	MoveL Offs(p0,555.9584000000001,76.2912, 0), v100, z5, tool0;
	MoveL Offs(p0,560.0348,77.80539999999999, 0), v100, z5, tool0;
	MoveL Offs(p0,563.6,79.4, 0), v100, z5, tool0;
	MoveL Offs(p0,569.7716,83.0468, 0), v100, z5, tool0;
	MoveL Offs(p0,575.6528000000001,87.57440000000001, 0), v100, z5, tool0;
	MoveL Offs(p0,581.1931999999999,92.90360000000001, 0), v100, z5, tool0;
	MoveL Offs(p0,586.3424,98.95520000000002, 0), v100, z5, tool0;
	MoveL Offs(p0,591.05,105.65, 0), v100, z5, tool0;
	MoveL Offs(p0,595.2656,112.9088, 0), v100, z5, tool0;
	MoveL Offs(p0,598.9388,120.65240000000001, 0), v100, z5, tool0;
	MoveL Offs(p0,602.0192000000001,128.8016, 0), v100, z5, tool0;
	MoveL Offs(p0,604.4564,137.27720000000002, 0), v100, z5, tool0;
	MoveL Offs(p0,606.2,146.0, 0), v100, z5, tool0;
	MoveL Offs(p0,607.3218,159.2564, 0), v100, z5, tool0;
	MoveL Offs(p0,606.7744000000002,172.87520000000006, 0), v100, z5, tool0;
	MoveL Offs(p0,604.6286,186.6908, 0), v100, z5, tool0;
	MoveL Offs(p0,600.9552,200.53760000000003, 0), v100, z5, tool0;
	MoveL Offs(p0,595.825,214.25, 0), v100, z5, tool0;
	MoveL Offs(p0,589.3088,227.66240000000002, 0), v100, z5, tool0;
	MoveL Offs(p0,581.4774,240.60919999999996, 0), v100, z5, tool0;
	MoveL Offs(p0,572.4015999999999,252.92480000000006, 0), v100, z5, tool0;
	MoveL Offs(p0,562.1522,264.4436, 0), v100, z5, tool0;
	MoveL Offs(p0,550.8,275.0, 0), v100, z5, tool0;
	MoveL Offs(p0,547.0016000000002,278.2064000000001, 0), v100, z5, tool0;
	MoveL Offs(p0,545.1804,279.7466, 0), v100, z5, tool0;
	MoveL Offs(p0,543.4528,281.21119999999996, 0), v100, z5, tool0;
	MoveL Offs(p0,541.85,282.575, 0), v100, z5, tool0;
	MoveL Offs(p0,540.4032,283.8128, 0), v100, z5, tool0;
	MoveL Offs(p0,539.1436,284.8994, 0), v100, z5, tool0;
	MoveL Offs(p0,538.1024,285.80960000000005, 0), v100, z5, tool0;
	MoveL Offs(p0,537.3108,286.51820000000004, 0), v100, z5, tool0;
	MoveL Offs(p0,536.8,287.0, 0), v100, z5, tool0;
	MoveL Offs(p0,534.559,288.72079999999994, 0), v100, z5, tool0;
	MoveL Offs(p0,533.376,289.6016, 0), v100, z5, tool0;
	MoveL Offs(p0,532.025,290.6, 0), v100, z5, tool0;
	MoveL Offs(p0,530.536,291.6944, 0), v100, z5, tool0;
	MoveL Offs(p0,528.939,292.86319999999995, 0), v100, z5, tool0;
	MoveL Offs(p0,527.264,294.0848, 0), v100, z5, tool0;
	MoveL Offs(p0,525.5409999999999,295.3376, 0), v100, z5, tool0;
	MoveL Offs(p0,523.8,296.6, 0), v100, z5, tool0;
	MoveL Offs(p0,518.3072,300.841, 0), v100, z5, tool0;
	MoveL Offs(p0,513.4576000000001,305.3040000000001, 0), v100, z5, tool0;
	MoveL Offs(p0,509.2344,310.019, 0), v100, z5, tool0;
	MoveL Offs(p0,505.62080000000003,315.016, 0), v100, z5, tool0;
	MoveL Offs(p0,502.6,320.325, 0), v100, z5, tool0;
	MoveL Offs(p0,500.1552,325.976, 0), v100, z5, tool0;
	MoveL Offs(p0,498.26959999999997,331.99899999999997, 0), v100, z5, tool0;
	MoveL Offs(p0,496.9264000000001,338.42400000000004, 0), v100, z5, tool0;
	MoveL Offs(p0,496.1088,345.281, 0), v100, z5, tool0;
	MoveL Offs(p0,495.8,352.6, 0), v100, z5, tool0;
	MoveL Offs(p0,495.9742,358.76900000000006, 0), v100, z5, tool0;
	MoveL Offs(p0,496.49760000000015,364.56000000000006, 0), v100, z5, tool0;
	MoveL Offs(p0,497.3714,369.979, 0), v100, z5, tool0;
	MoveL Offs(p0,498.5968,375.03200000000004, 0), v100, z5, tool0;
	MoveL Offs(p0,500.175,379.725, 0), v100, z5, tool0;
	MoveL Offs(p0,502.10720000000003,384.06399999999996, 0), v100, z5, tool0;
	MoveL Offs(p0,504.39459999999997,388.055, 0), v100, z5, tool0;
	MoveL Offs(p0,507.0384,391.704, 0), v100, z5, tool0;
	MoveL Offs(p0,510.0398,395.017, 0), v100, z5, tool0;
	MoveL Offs(p0,513.4,398.0, 0), v100, z5, tool0;
	MoveL Offs(p0,516.6784000000001,400.3968000000001, 0), v100, z5, tool0;
	MoveL Offs(p0,517.9666,401.13919999999996, 0), v100, z5, tool0;
	MoveL Offs(p0,519.0832,401.5744000000001, 0), v100, z5, tool0;
	MoveL Offs(p0,520.075,401.7, 0), v100, z5, tool0;
	MoveL Offs(p0,520.9888,401.51360000000005, 0), v100, z5, tool0;
	MoveL Offs(p0,521.8714,401.01279999999997, 0), v100, z5, tool0;
	MoveL Offs(p0,522.7696,400.1952, 0), v100, z5, tool0;
	MoveL Offs(p0,523.7302,399.0584, 0), v100, z5, tool0;
	MoveL Offs(p0,524.8,397.6, 0), v100, z5, tool0;
	MoveL Offs(p0,524.8,397.6, 0), v100, z5, tool0;
	MoveJ Offs(p0,74.2,395.8, 10), v100, z1, tool0;
	MoveL Offs(p0,76.83040000000003,394.7840000000001, 0), v100, z5, tool0;
	MoveL Offs(p0,78.1906,394.162, 0), v100, z5, tool0;
	MoveL Offs(p0,79.5472,393.47999999999996, 0), v100, z5, tool0;
	MoveL Offs(p0,80.875,392.75, 0), v100, z5, tool0;
	MoveL Offs(p0,82.14880000000001,391.984, 0), v100, z5, tool0;
	MoveL Offs(p0,83.3434,391.194, 0), v100, z5, tool0;
	MoveL Offs(p0,84.4336,390.392, 0), v100, z5, tool0;
	MoveL Offs(p0,85.3942,389.59000000000003, 0), v100, z5, tool0;
	MoveL Offs(p0,86.2,388.8, 0), v100, z5, tool0;
	MoveL Offs(p0,90.4,384.4, 0), v100, z5, tool0;
	MoveL Offs(p0,81.6,373.6, 0), v100, z5, tool0;
	MoveL Offs(p0,78.64320000000002,369.6352000000001, 0), v100, z5, tool0;
	MoveL Offs(p0,77.0658,367.36479999999995, 0), v100, z5, tool0;
	MoveL Offs(p0,75.46560000000001,364.9696, 0), v100, z5, tool0;
	MoveL Offs(p0,73.875,362.5, 0), v100, z5, tool0;
	MoveL Offs(p0,72.32639999999999,360.0064, 0), v100, z5, tool0;
	MoveL Offs(p0,70.85220000000001,357.5392, 0), v100, z5, tool0;
	MoveL Offs(p0,69.4848,355.14880000000005, 0), v100, z5, tool0;
	MoveL Offs(p0,68.2566,352.8856, 0), v100, z5, tool0;
	MoveL Offs(p0,67.2,350.8, 0), v100, z5, tool0;
	MoveL Offs(p0,65.66760000000001,347.5358, 0), v100, z5, tool0;
	MoveL Offs(p0,64.37280000000001,344.8944000000001, 0), v100, z5, tool0;
	MoveL Offs(p0,63.229200000000006,342.8026, 0), v100, z5, tool0;
	MoveL Offs(p0,62.150400000000005,341.1872, 0), v100, z5, tool0;
	MoveL Offs(p0,61.05,339.975, 0), v100, z5, tool0;
	MoveL Offs(p0,59.84159999999999,339.0928, 0), v100, z5, tool0;
	MoveL Offs(p0,58.43879999999999,338.4674, 0), v100, z5, tool0;
	MoveL Offs(p0,56.755200000000016,338.02560000000005, 0), v100, z5, tool0;
	MoveL Offs(p0,54.70440000000001,337.6942, 0), v100, z5, tool0;
	MoveL Offs(p0,52.2,337.4, 0), v100, z5, tool0;
	MoveL Offs(p0,49.16320000000002,336.9968000000001, 0), v100, z5, tool0;
	MoveL Offs(p0,47.6568,336.7682, 0), v100, z5, tool0;
	MoveL Offs(p0,46.1936,336.5264000000001, 0), v100, z5, tool0;
	MoveL Offs(p0,44.8,336.275, 0), v100, z5, tool0;
	MoveL Offs(p0,43.5024,336.0176, 0), v100, z5, tool0;
	MoveL Offs(p0,42.32719999999999,335.7578, 0), v100, z5, tool0;
	MoveL Offs(p0,41.3008,335.49920000000003, 0), v100, z5, tool0;
	MoveL Offs(p0,40.449600000000004,335.24539999999996, 0), v100, z5, tool0;
	MoveL Offs(p0,39.8,335.0, 0), v100, z5, tool0;
	MoveL Offs(p0,37.342400000000005,336.648, 0), v100, z5, tool0;
	MoveL Offs(p0,36.95,338.35, 0), v100, z5, tool0;
	MoveL Offs(p0,36.6176,340.76, 0), v100, z5, tool0;
	MoveL Offs(p0,36.330799999999996,343.974, 0), v100, z5, tool0;
	MoveL Offs(p0,36.07520000000001,348.088, 0), v100, z5, tool0;
	MoveL Offs(p0,35.836400000000005,353.198, 0), v100, z5, tool0;
	MoveL Offs(p0,35.6,359.4, 0), v100, z5, tool0;
	MoveL Offs(p0,35.343,365.43420000000003, 0), v100, z5, tool0;
	MoveL Offs(p0,35.17600000000001,370.52160000000003, 0), v100, z5, tool0;
	MoveL Offs(p0,35.105,374.7594, 0), v100, z5, tool0;
	MoveL Offs(p0,35.136,378.2448, 0), v100, z5, tool0;
	MoveL Offs(p0,35.275,381.075, 0), v100, z5, tool0;
	MoveL Offs(p0,35.528,383.34720000000004, 0), v100, z5, tool0;
	MoveL Offs(p0,35.900999999999996,385.1586, 0), v100, z5, tool0;
	MoveL Offs(p0,36.400000000000006,386.6064, 0), v100, z5, tool0;
	MoveL Offs(p0,37.031,387.7878, 0), v100, z5, tool0;
	MoveL Offs(p0,37.8,388.8, 0), v100, z5, tool0;
	MoveL Offs(p0,40.223200000000006,391.15060000000005, 0), v100, z5, tool0;
	MoveL Offs(p0,43.02560000000001,393.1568000000001, 0), v100, z5, tool0;
	MoveL Offs(p0,46.166399999999996,394.8102, 0), v100, z5, tool0;
	MoveL Offs(p0,49.6048,396.10240000000005, 0), v100, z5, tool0;
	MoveL Offs(p0,53.3,397.025, 0), v100, z5, tool0;
	MoveL Offs(p0,57.2112,397.5696, 0), v100, z5, tool0;
	MoveL Offs(p0,61.2976,397.72779999999995, 0), v100, z5, tool0;
	MoveL Offs(p0,65.51840000000001,397.49120000000005, 0), v100, z5, tool0;
	MoveL Offs(p0,69.8328,396.8514, 0), v100, z5, tool0;
	MoveL Offs(p0,74.2,395.8, 0), v100, z5, tool0;
	MoveL Offs(p0,74.2,395.8, 0), v100, z5, tool0;
	MoveJ Offs(p0,31.6,355.4, 10), v100, z1, tool0;
	MoveL Offs(p0,31.0,330.8, 0), v100, z5, tool0;
	MoveL Offs(p0,24.0,324.6, 0), v100, z5, tool0;
	MoveL Offs(p0,17.0,318.2, 0), v100, z5, tool0;
	MoveL Offs(p0,15.6,324.6, 0), v100, z5, tool0;
	MoveL Offs(p0,15.240000000000004,327.3088000000001, 0), v100, z5, tool0;
	MoveL Offs(p0,15.149999999999997,329.0172, 0), v100, z5, tool0;
	MoveL Offs(p0,15.12,330.91040000000004, 0), v100, z5, tool0;
	MoveL Offs(p0,15.15,332.95, 0), v100, z5, tool0;
	MoveL Offs(p0,15.24,335.0976, 0), v100, z5, tool0;
	MoveL Offs(p0,15.39,337.3148, 0), v100, z5, tool0;
	MoveL Offs(p0,15.6,339.56320000000005, 0), v100, z5, tool0;
	MoveL Offs(p0,15.87,341.8044, 0), v100, z5, tool0;
	MoveL Offs(p0,16.2,344.0, 0), v100, z5, tool0;
	MoveL Offs(p0,17.0458,348.31280000000004, 0), v100, z5, tool0;
	MoveL Offs(p0,18.214400000000005,352.96640000000014, 0), v100, z5, tool0;
	MoveL Offs(p0,19.6326,357.7736, 0), v100, z5, tool0;
	MoveL Offs(p0,21.227200000000003,362.5472, 0), v100, z5, tool0;
	MoveL Offs(p0,22.925,367.1, 0), v100, z5, tool0;
	MoveL Offs(p0,24.652800000000003,371.24479999999994, 0), v100, z5, tool0;
	MoveL Offs(p0,26.337400000000002,374.79440000000005, 0), v100, z5, tool0;
	MoveL Offs(p0,27.905600000000003,377.5616, 0), v100, z5, tool0;
	MoveL Offs(p0,29.284200000000006,379.3592, 0), v100, z5, tool0;
	MoveL Offs(p0,30.4,380.0, 0), v100, z5, tool0;
	MoveL Offs(p0,31.264,377.4458, 0), v100, z5, tool0;
	MoveL Offs(p0,31.456,375.54560000000004, 0), v100, z5, tool0;
	MoveL Offs(p0,31.6,373.175, 0), v100, z5, tool0;
	MoveL Offs(p0,31.696000000000005,370.3664, 0), v100, z5, tool0;
	MoveL Offs(p0,31.744,367.1522, 0), v100, z5, tool0;
	MoveL Offs(p0,31.744,363.5648, 0), v100, z5, tool0;
	MoveL Offs(p0,31.696000000000005,359.63660000000004, 0), v100, z5, tool0;
	MoveL Offs(p0,31.6,355.4, 0), v100, z5, tool0;
	MoveL Offs(p0,31.6,355.4, 0), v100, z5, tool0;
	MoveJ Offs(p0,94.0,373.8, 10), v100, z1, tool0;
	MoveL Offs(p0,93.85920000000002,371.1684, 0), v100, z5, tool0;
	MoveL Offs(p0,93.44960000000003,368.3472000000001, 0), v100, z5, tool0;
	MoveL Offs(p0,92.7904,365.3868, 0), v100, z5, tool0;
	MoveL Offs(p0,91.9008,362.3376, 0), v100, z5, tool0;
	MoveL Offs(p0,90.8,359.25, 0), v100, z5, tool0;
	MoveL Offs(p0,89.5072,356.1744, 0), v100, z5, tool0;
	MoveL Offs(p0,88.04159999999999,353.1612, 0), v100, z5, tool0;
	MoveL Offs(p0,86.42240000000001,350.2608, 0), v100, z5, tool0;
	MoveL Offs(p0,84.6688,347.5236, 0), v100, z5, tool0;
	MoveL Offs(p0,82.8,345.0, 0), v100, z5, tool0;
	MoveL Offs(p0,79.81880000000001,341.09479999999996, 0), v100, z5, tool0;
	MoveL Offs(p0,77.47840000000001,337.80640000000005, 0), v100, z5, tool0;
	MoveL Offs(p0,75.78359999999999,335.1756, 0), v100, z5, tool0;
	MoveL Offs(p0,74.73920000000001,333.2432, 0), v100, z5, tool0;
	MoveL Offs(p0,74.35,332.05, 0), v100, z5, tool0;
	MoveL Offs(p0,74.6208,331.6368, 0), v100, z5, tool0;
	MoveL Offs(p0,75.55640000000001,332.04440000000005, 0), v100, z5, tool0;
	MoveL Offs(p0,77.16159999999999,333.31360000000006, 0), v100, z5, tool0;
	MoveL Offs(p0,79.44120000000001,335.48519999999996, 0), v100, z5, tool0;
	MoveL Offs(p0,82.4,338.6, 0), v100, z5, tool0;
	MoveL Offs(p0,85.2108,341.66740000000004, 0), v100, z5, tool0;
	MoveL Offs(p0,87.65440000000002,344.1552000000001, 0), v100, z5, tool0;
	MoveL Offs(p0,89.7476,346.0718, 0), v100, z5, tool0;
	MoveL Offs(p0,91.50720000000001,347.42560000000003, 0), v100, z5, tool0;
	MoveL Offs(p0,92.95,348.225, 0), v100, z5, tool0;
	MoveL Offs(p0,94.0928,348.4784, 0), v100, z5, tool0;
	MoveL Offs(p0,94.9524,348.19419999999997, 0), v100, z5, tool0;
	MoveL Offs(p0,95.54560000000001,347.3808, 0), v100, z5, tool0;
	MoveL Offs(p0,95.8892,346.0466, 0), v100, z5, tool0;
	MoveL Offs(p0,96.0,344.2, 0), v100, z5, tool0;
	MoveL Offs(p0,95.54020000000001,341.5576, 0), v100, z5, tool0;
	MoveL Offs(p0,94.26560000000003,337.89280000000014, 0), v100, z5, tool0;
	MoveL Offs(p0,92.33339999999998,333.47920000000005, 0), v100, z5, tool0;
	MoveL Offs(p0,89.9008,328.5904, 0), v100, z5, tool0;
	MoveL Offs(p0,87.125,323.5, 0), v100, z5, tool0;
	MoveL Offs(p0,84.16319999999999,318.48159999999996, 0), v100, z5, tool0;
	MoveL Offs(p0,81.1726,313.80879999999996, 0), v100, z5, tool0;
	MoveL Offs(p0,78.3104,309.7552, 0), v100, z5, tool0;
	MoveL Offs(p0,75.7338,306.5944, 0), v100, z5, tool0;
	MoveL Offs(p0,73.6,304.6, 0), v100, z5, tool0;
	MoveL Offs(p0,71.49920000000002,303.0282, 0), v100, z5, tool0;
	MoveL Offs(p0,70.08960000000002,301.7936, 0), v100, z5, tool0;
	MoveL Offs(p0,69.33040000000001,300.8974, 0), v100, z5, tool0;
	MoveL Offs(p0,69.1808,300.34080000000006, 0), v100, z5, tool0;
	MoveL Offs(p0,69.6,300.125, 0), v100, z5, tool0;
	MoveL Offs(p0,70.5472,300.2512, 0), v100, z5, tool0;
	MoveL Offs(p0,71.9816,300.7206, 0), v100, z5, tool0;
	MoveL Offs(p0,73.86240000000001,301.5344, 0), v100, z5, tool0;
	MoveL Offs(p0,76.14880000000001,302.6938, 0), v100, z5, tool0;
	MoveL Offs(p0,78.8,304.2, 0), v100, z5, tool0;
	MoveL Offs(p0,82.03520000000003,306.03040000000004, 0), v100, z5, tool0;
	MoveL Offs(p0,83.2478,306.6156, 0), v100, z5, tool0;
	MoveL Offs(p0,84.2336,306.98720000000003, 0), v100, z5, tool0;
	MoveL Offs(p0,85.025,307.15, 0), v100, z5, tool0;
	MoveL Offs(p0,85.65440000000001,307.1088, 0), v100, z5, tool0;
	MoveL Offs(p0,86.15419999999999,306.8684, 0), v100, z5, tool0;
	MoveL Offs(p0,86.5568,306.4336, 0), v100, z5, tool0;
	MoveL Offs(p0,86.89460000000001,305.80920000000003, 0), v100, z5, tool0;
	MoveL Offs(p0,87.2,305.0, 0), v100, z5, tool0;
	MoveL Offs(p0,87.48640000000002,302.431, 0), v100, z5, tool0;
	MoveL Offs(p0,86.77920000000003,299.0880000000001, 0), v100, z5, tool0;
	MoveL Offs(p0,85.24879999999999,295.217, 0), v100, z5, tool0;
	MoveL Offs(p0,83.0656,291.064, 0), v100, z5, tool0;
	MoveL Offs(p0,80.4,286.875, 0), v100, z5, tool0;
	MoveL Offs(p0,77.42240000000001,282.896, 0), v100, z5, tool0;
	MoveL Offs(p0,74.3032,279.373, 0), v100, z5, tool0;
	MoveL Offs(p0,71.2128,276.552, 0), v100, z5, tool0;
	MoveL Offs(p0,68.3216,274.679, 0), v100, z5, tool0;
	MoveL Offs(p0,65.8,274.0, 0), v100, z5, tool0;
	MoveL Offs(p0,63.11040000000003,275.6784000000001, 0), v100, z5, tool0;
	MoveL Offs(p0,61.9336,277.6666, 0), v100, z5, tool0;
	MoveL Offs(p0,60.891200000000005,280.3232, 0), v100, z5, tool0;
	MoveL Offs(p0,60.0,283.575, 0), v100, z5, tool0;
	MoveL Offs(p0,59.2768,287.3488, 0), v100, z5, tool0;
	MoveL Offs(p0,58.73839999999999,291.5714, 0), v100, z5, tool0;
	MoveL Offs(p0,58.40160000000001,296.1696, 0), v100, z5, tool0;
	MoveL Offs(p0,58.2832,301.0702, 0), v100, z5, tool0;
	MoveL Offs(p0,58.4,306.2, 0), v100, z5, tool0;
	MoveL Offs(p0,58.65200000000001,310.39740000000006, 0), v100, z5, tool0;
	MoveL Offs(p0,58.95200000000002,314.0752000000001, 0), v100, z5, tool0;
	MoveL Offs(p0,59.336,317.3618, 0), v100, z5, tool0;
	MoveL Offs(p0,59.84000000000001,320.3856, 0), v100, z5, tool0;
	MoveL Offs(p0,60.5,323.275, 0), v100, z5, tool0;
	MoveL Offs(p0,61.352,326.1584, 0), v100, z5, tool0;
	MoveL Offs(p0,62.432,329.1642, 0), v100, z5, tool0;
	MoveL Offs(p0,63.775999999999996,332.42080000000004, 0), v100, z5, tool0;
	MoveL Offs(p0,65.42,336.0566, 0), v100, z5, tool0;
	MoveL Offs(p0,67.4,340.2, 0), v100, z5, tool0;
	MoveL Offs(p0,70.04920000000001,345.5352000000001, 0), v100, z5, tool0;
	MoveL Offs(p0,72.89760000000003,350.8896000000001, 0), v100, z5, tool0;
	MoveL Offs(p0,75.8564,356.1264, 0), v100, z5, tool0;
	MoveL Offs(p0,78.83680000000001,361.1088000000001, 0), v100, z5, tool0;
	MoveL Offs(p0,81.75,365.7, 0), v100, z5, tool0;
	MoveL Offs(p0,84.50720000000001,369.7632, 0), v100, z5, tool0;
	MoveL Offs(p0,87.0196,373.1616, 0), v100, z5, tool0;
	MoveL Offs(p0,89.19840000000002,375.75840000000005, 0), v100, z5, tool0;
	MoveL Offs(p0,90.9548,377.4168, 0), v100, z5, tool0;
	MoveL Offs(p0,92.2,378.0, 0), v100, z5, tool0;
	MoveL Offs(p0,93.80019999999999,375.67740000000003, 0), v100, z5, tool0;
	MoveL Offs(p0,93.9088,375.0816, 0), v100, z5, tool0;
	MoveL Offs(p0,93.9766,374.4522, 0), v100, z5, tool0;
	MoveL Offs(p0,94.0,373.8, 0), v100, z5, tool0;
	MoveL Offs(p0,94.0,373.8, 0), v100, z5, tool0;
	MoveJ Offs(p0,490.2,367.2, 10), v100, z1, tool0;
	MoveL Offs(p0,489.338,360.44860000000006, 0), v100, z5, tool0;
	MoveL Offs(p0,489.1360000000001,353.4608000000001, 0), v100, z5, tool0;
	MoveL Offs(p0,489.57,346.33619999999996, 0), v100, z5, tool0;
	MoveL Offs(p0,490.6160000000001,339.1744, 0), v100, z5, tool0;
	MoveL Offs(p0,492.25,332.075, 0), v100, z5, tool0;
	MoveL Offs(p0,494.448,325.13759999999996, 0), v100, z5, tool0;
	MoveL Offs(p0,497.186,318.4618, 0), v100, z5, tool0;
	MoveL Offs(p0,500.44000000000005,312.1472, 0), v100, z5, tool0;
	MoveL Offs(p0,504.18600000000004,306.2934, 0), v100, z5, tool0;
	MoveL Offs(p0,508.4,301.0, 0), v100, z5, tool0;
	MoveL Offs(p0,514.6,293.8, 0), v100, z5, tool0;
	MoveL Offs(p0,505.8,284.8, 0), v100, z5, tool0;
	MoveL Offs(p0,500.2146000000001,279.73580000000004, 0), v100, z5, tool0;
	MoveL Offs(p0,493.85280000000023,275.1264000000001, 0), v100, z5, tool0;
	MoveL Offs(p0,486.8262,271.00660000000005, 0), v100, z5, tool0;
	MoveL Offs(p0,479.2464000000001,267.4112, 0), v100, z5, tool0;
	MoveL Offs(p0,471.225,264.375, 0), v100, z5, tool0;
	MoveL Offs(p0,462.8736,261.9328, 0), v100, z5, tool0;
	MoveL Offs(p0,454.30379999999997,260.1194, 0), v100, z5, tool0;
	MoveL Offs(p0,445.6272000000001,258.9696, 0), v100, z5, tool0;
	MoveL Offs(p0,436.9554,258.51820000000004, 0), v100, z5, tool0;
	MoveL Offs(p0,428.4,258.8, 0), v100, z5, tool0;
	MoveL Offs(p0,423.1018,259.3242, 0), v100, z5, tool0;
	MoveL Offs(p0,418.2224000000001,260.0656000000001, 0), v100, z5, tool0;
	MoveL Offs(p0,413.7246,261.0374, 0), v100, z5, tool0;
	MoveL Offs(p0,409.5712,262.2528, 0), v100, z5, tool0;
	MoveL Offs(p0,405.725,263.725, 0), v100, z5, tool0;
	MoveL Offs(p0,402.1488,265.46719999999993, 0), v100, z5, tool0;
	MoveL Offs(p0,398.8054,267.4926, 0), v100, z5, tool0;
	MoveL Offs(p0,395.65760000000006,269.81440000000003, 0), v100, z5, tool0;
	MoveL Offs(p0,392.66819999999996,272.4458, 0), v100, z5, tool0;
	MoveL Offs(p0,389.8,275.4, 0), v100, z5, tool0;
	MoveL Offs(p0,387.26020000000005,278.356, 0), v100, z5, tool0;
	MoveL Offs(p0,385.0336000000001,281.36, 0), v100, z5, tool0;
	MoveL Offs(p0,383.1094,284.436, 0), v100, z5, tool0;
	MoveL Offs(p0,381.4768,287.608, 0), v100, z5, tool0;
	MoveL Offs(p0,380.125,290.9, 0), v100, z5, tool0;
	MoveL Offs(p0,379.04319999999996,294.33599999999996, 0), v100, z5, tool0;
	MoveL Offs(p0,378.2206,297.93999999999994, 0), v100, z5, tool0;
	MoveL Offs(p0,377.64639999999997,301.736, 0), v100, z5, tool0;
	MoveL Offs(p0,377.30980000000005,305.748, 0), v100, z5, tool0;
	MoveL Offs(p0,377.2,310.0, 0), v100, z5, tool0;
	MoveL Offs(p0,377.43420000000003,314.0904, 0), v100, z5, tool0;
	MoveL Offs(p0,378.0896000000001,318.55520000000007, 0), v100, z5, tool0;
	MoveL Offs(p0,379.0954,323.20480000000003, 0), v100, z5, tool0;
	MoveL Offs(p0,380.3808,327.8496, 0), v100, z5, tool0;
	MoveL Offs(p0,381.875,332.3, 0), v100, z5, tool0;
	MoveL Offs(p0,383.5072,336.3664, 0), v100, z5, tool0;
	MoveL Offs(p0,385.2066,339.8592, 0), v100, z5, tool0;
	MoveL Offs(p0,386.90240000000006,342.5888, 0), v100, z5, tool0;
	MoveL Offs(p0,388.52380000000005,344.3656, 0), v100, z5, tool0;
	MoveL Offs(p0,390.0,345.0, 0), v100, z5, tool0;
	MoveL Offs(p0,392.59200000000004,343.27200000000005, 0), v100, z5, tool0;
	MoveL Offs(p0,393.375,342.375, 0), v100, z5, tool0;
	MoveL Offs(p0,394.17600000000004,341.328, 0), v100, z5, tool0;
	MoveL Offs(p0,394.97700000000003,340.149, 0), v100, z5, tool0;
	MoveL Offs(p0,395.76000000000005,338.85600000000005, 0), v100, z5, tool0;
	MoveL Offs(p0,396.50699999999995,337.467, 0), v100, z5, tool0;
	MoveL Offs(p0,397.2,336.0, 0), v100, z5, tool0;
	MoveL Offs(p0,399.08660000000003,332.43420000000003, 0), v100, z5, tool0;
	MoveL Offs(p0,401.03680000000014,329.2896000000001, 0), v100, z5, tool0;
	MoveL Offs(p0,403.0661999999999,326.5554, 0), v100, z5, tool0;
	MoveL Offs(p0,405.1904,324.2208, 0), v100, z5, tool0;
	MoveL Offs(p0,407.425,322.275, 0), v100, z5, tool0;
	MoveL Offs(p0,409.7856,320.7072, 0), v100, z5, tool0;
	MoveL Offs(p0,412.28779999999995,319.50660000000005, 0), v100, z5, tool0;
	MoveL Offs(p0,414.94719999999995,318.66240000000005, 0), v100, z5, tool0;
	MoveL Offs(p0,417.7794,318.1638, 0), v100, z5, tool0;
	MoveL Offs(p0,420.8,318.0, 0), v100, z5, tool0;
	MoveL Offs(p0,423.5510000000001,318.04460000000006, 0), v100, z5, tool0;
	MoveL Offs(p0,425.8880000000001,318.26080000000013, 0), v100, z5, tool0;
	MoveL Offs(p0,427.937,318.7722, 0), v100, z5, tool0;
	MoveL Offs(p0,429.82400000000007,319.70240000000007, 0), v100, z5, tool0;
	MoveL Offs(p0,431.675,321.175, 0), v100, z5, tool0;
	MoveL Offs(p0,433.616,323.3136, 0), v100, z5, tool0;
	MoveL Offs(p0,435.773,326.24179999999996, 0), v100, z5, tool0;
	MoveL Offs(p0,438.2720000000001,330.08320000000003, 0), v100, z5, tool0;
	MoveL Offs(p0,441.23900000000003,334.9614, 0), v100, z5, tool0;
	MoveL Offs(p0,444.8,341.0, 0), v100, z5, tool0;
	MoveL Offs(p0,447.23580000000004,345.10940000000005, 0), v100, z5, tool0;
	MoveL Offs(p0,449.3344000000001,348.5072000000001, 0), v100, z5, tool0;
	MoveL Offs(p0,451.20259999999996,351.2978, 0), v100, z5, tool0;
	MoveL Offs(p0,452.94720000000007,353.5856, 0), v100, z5, tool0;
	MoveL Offs(p0,454.675,355.475, 0), v100, z5, tool0;
	MoveL Offs(p0,456.4928,357.07039999999995, 0), v100, z5, tool0;
	MoveL Offs(p0,458.50739999999996,358.4762, 0), v100, z5, tool0;
	MoveL Offs(p0,460.8256,359.79679999999996, 0), v100, z5, tool0;
	MoveL Offs(p0,463.5541999999999,361.1366, 0), v100, z5, tool0;
	MoveL Offs(p0,466.8,362.6, 0), v100, z5, tool0;
	MoveL Offs(p0,468.87560000000013,363.55000000000007, 0), v100, z5, tool0;
	MoveL Offs(p0,470.9968000000002,364.5840000000002, 0), v100, z5, tool0;
	MoveL Offs(p0,473.12519999999995,365.678, 0), v100, z5, tool0;
	MoveL Offs(p0,475.2224,366.8080000000001, 0), v100, z5, tool0;
	MoveL Offs(p0,477.25,367.95, 0), v100, z5, tool0;
	MoveL Offs(p0,479.1696,369.08, 0), v100, z5, tool0;
	MoveL Offs(p0,480.9428,370.174, 0), v100, z5, tool0;
	MoveL Offs(p0,482.53120000000007,371.20799999999997, 0), v100, z5, tool0;
	MoveL Offs(p0,483.89639999999997,372.158, 0), v100, z5, tool0;
	MoveL Offs(p0,485.0,373.0, 0), v100, z5, tool0;
	MoveL Offs(p0,487.84939999999995,375.09159999999997, 0), v100, z5, tool0;
	MoveL Offs(p0,488.6768,375.6592, 0), v100, z5, tool0;
	MoveL Offs(p0,489.425,376.15, 0), v100, z5, tool0;
	MoveL Offs(p0,490.08320000000003,376.55679999999995, 0), v100, z5, tool0;
	MoveL Offs(p0,490.6406,376.8724, 0), v100, z5, tool0;
	MoveL Offs(p0,491.0864,377.0896000000001, 0), v100, z5, tool0;
	MoveL Offs(p0,491.4098,377.20120000000003, 0), v100, z5, tool0;
	MoveL Offs(p0,491.6,377.2, 0), v100, z5, tool0;
	MoveL Offs(p0,491.48159999999996,375.00480000000005, 0), v100, z5, tool0;
	MoveL Offs(p0,491.35,374.0, 0), v100, z5, tool0;
	MoveL Offs(p0,491.1824,372.8512, 0), v100, z5, tool0;
	MoveL Offs(p0,490.9812,371.57759999999996, 0), v100, z5, tool0;
	MoveL Offs(p0,490.7488,370.19840000000005, 0), v100, z5, tool0;
	MoveL Offs(p0,490.48760000000004,368.73280000000005, 0), v100, z5, tool0;
	MoveL Offs(p0,490.2,367.2, 0), v100, z5, tool0;
	MoveL Offs(p0,490.2,367.2, 0), v100, z5, tool0;
	MoveJ Offs(p0,524.2,363.6, 10), v100, z1, tool0;
	MoveL Offs(p0,524.865,359.97120000000007, 0), v100, z5, tool0;
	MoveL Offs(p0,525.416,355.4016000000001, 0), v100, z5, tool0;
	MoveL Offs(p0,525.847,350.18639999999994, 0), v100, z5, tool0;
	MoveL Offs(p0,526.152,344.62080000000003, 0), v100, z5, tool0;
	MoveL Offs(p0,526.325,339.0, 0), v100, z5, tool0;
	MoveL Offs(p0,526.36,333.6192, 0), v100, z5, tool0;
	MoveL Offs(p0,526.251,328.7736, 0), v100, z5, tool0;
	MoveL Offs(p0,525.992,324.75840000000005, 0), v100, z5, tool0;
	MoveL Offs(p0,525.577,321.8688, 0), v100, z5, tool0;
	MoveL Offs(p0,525.0,320.4, 0), v100, z5, tool0;
	MoveL Offs(p0,522.5196,321.1974, 0), v100, z5, tool0;
	MoveL Offs(p0,521.4671999999999,322.4928, 0), v100, z5, tool0;
	MoveL Offs(p0,520.35,324.225, 0), v100, z5, tool0;
	MoveL Offs(p0,519.1967999999999,326.3472, 0), v100, z5, tool0;
	MoveL Offs(p0,518.0364,328.81260000000003, 0), v100, z5, tool0;
	MoveL Offs(p0,516.8976,331.5744000000001, 0), v100, z5, tool0;
	MoveL Offs(p0,515.8092,334.5858, 0), v100, z5, tool0;
	MoveL Offs(p0,514.8,337.8, 0), v100, z5, tool0;
	MoveL Offs(p0,513.894,341.11080000000004, 0), v100, z5, tool0;
	MoveL Offs(p0,513.2160000000001,344.4384000000001, 0), v100, z5, tool0;
	MoveL Offs(p0,512.766,347.77560000000005, 0), v100, z5, tool0;
	MoveL Offs(p0,512.544,351.1152, 0), v100, z5, tool0;
	MoveL Offs(p0,512.55,354.45, 0), v100, z5, tool0;
	MoveL Offs(p0,512.784,357.7728, 0), v100, z5, tool0;
	MoveL Offs(p0,513.246,361.07640000000004, 0), v100, z5, tool0;
	MoveL Offs(p0,513.936,364.35360000000003, 0), v100, z5, tool0;
	MoveL Offs(p0,514.854,367.59720000000004, 0), v100, z5, tool0;
	MoveL Offs(p0,516.0,370.8, 0), v100, z5, tool0;
	MoveL Offs(p0,517.6208,374.08320000000015, 0), v100, z5, tool0;
	MoveL Offs(p0,518.4012,374.85179999999997, 0), v100, z5, tool0;
	MoveL Offs(p0,519.1744000000001,375.0336000000001, 0), v100, z5, tool0;
	MoveL Offs(p0,519.95,374.625, 0), v100, z5, tool0;
	MoveL Offs(p0,520.7376,373.6224, 0), v100, z5, tool0;
	MoveL Offs(p0,521.5468,372.0222, 0), v100, z5, tool0;
	MoveL Offs(p0,522.3872,369.8208000000001, 0), v100, z5, tool0;
	MoveL Offs(p0,523.2684,367.0146, 0), v100, z5, tool0;
	MoveL Offs(p0,524.2,363.6, 0), v100, z5, tool0;
	MoveL Offs(p0,524.2,363.6, 0), v100, z5, tool0;
	MoveJ Offs(p0,95.4,355.6, 10), v100, z1, tool0;
	MoveL Offs(p0,94.2928,358.8960000000001, 0), v100, z5, tool0;
	MoveL Offs(p0,94.4,359.225, 0), v100, z5, tool0;
	MoveL Offs(p0,94.53119999999998,359.464, 0), v100, z5, tool0;
	MoveL Offs(p0,94.68159999999999,359.60699999999997, 0), v100, z5, tool0;
	MoveL Offs(p0,94.8464,359.648, 0), v100, z5, tool0;
	MoveL Offs(p0,95.0208,359.581, 0), v100, z5, tool0;
	MoveL Offs(p0,95.2,359.4, 0), v100, z5, tool0;
	MoveL Offs(p0,95.7616,357.3696, 0), v100, z5, tool0;
	MoveL Offs(p0,95.7348,356.92480000000006, 0), v100, z5, tool0;
	MoveL Offs(p0,95.66720000000001,356.47520000000003, 0), v100, z5, tool0;
	MoveL Offs(p0,95.55640000000001,356.0304, 0), v100, z5, tool0;
	MoveL Offs(p0,95.4,355.6, 0), v100, z5, tool0;
	MoveL Offs(p0,95.4,355.6, 0), v100, z5, tool0;
	MoveJ Offs(p0,352.4,341.6, 10), v100, z1, tool0;
	MoveL Offs(p0,352.32120000000003,339.33340000000004, 0), v100, z5, tool0;
	MoveL Offs(p0,352.3216000000001,336.8832000000001, 0), v100, z5, tool0;
	MoveL Offs(p0,352.39639999999997,334.29380000000003, 0), v100, z5, tool0;
	MoveL Offs(p0,352.5408,331.6096, 0), v100, z5, tool0;
	MoveL Offs(p0,352.75,328.875, 0), v100, z5, tool0;
	MoveL Offs(p0,353.0192,326.1344, 0), v100, z5, tool0;
	MoveL Offs(p0,353.3436,323.4322, 0), v100, z5, tool0;
	MoveL Offs(p0,353.71840000000003,320.81280000000004, 0), v100, z5, tool0;
	MoveL Offs(p0,354.1388,318.3206, 0), v100, z5, tool0;
	MoveL Offs(p0,354.6,316.0, 0), v100, z5, tool0;
	MoveL Offs(p0,355.4864,312.1186000000001, 0), v100, z5, tool0;
	MoveL Offs(p0,356.0992000000001,308.8528, 0), v100, z5, tool0;
	MoveL Offs(p0,356.4288,306.17019999999997, 0), v100, z5, tool0;
	MoveL Offs(p0,356.4656,304.0384, 0), v100, z5, tool0;
	MoveL Offs(p0,356.2,302.425, 0), v100, z5, tool0;
	MoveL Offs(p0,355.62239999999997,301.2976, 0), v100, z5, tool0;
	MoveL Offs(p0,354.7232,300.6238, 0), v100, z5, tool0;
	MoveL Offs(p0,353.49280000000005,300.37120000000004, 0), v100, z5, tool0;
	MoveL Offs(p0,351.9216,300.5074000000001, 0), v100, z5, tool0;
	MoveL Offs(p0,350.0,301.0, 0), v100, z5, tool0;
	MoveL Offs(p0,346.91280000000006,302.78080000000006, 0), v100, z5, tool0;
	MoveL Offs(p0,343.6384000000001,305.98240000000004, 0), v100, z5, tool0;
	MoveL Offs(p0,340.33759999999995,310.2736, 0), v100, z5, tool0;
	MoveL Offs(p0,337.17120000000006,315.32320000000004, 0), v100, z5, tool0;
	MoveL Offs(p0,334.3,320.8, 0), v100, z5, tool0;
	MoveL Offs(p0,331.8848,326.3728, 0), v100, z5, tool0;
	MoveL Offs(p0,330.0864,331.7104, 0), v100, z5, tool0;
	MoveL Offs(p0,329.0656,336.4816, 0), v100, z5, tool0;
	MoveL Offs(p0,328.9832,340.3552, 0), v100, z5, tool0;
	MoveL Offs(p0,330.0,343.0, 0), v100, z5, tool0;
	MoveL Offs(p0,332.7984,345.2960000000001, 0), v100, z5, tool0;
	MoveL Offs(p0,334.9896,346.69899999999996, 0), v100, z5, tool0;
	MoveL Offs(p0,337.5072,348.168, 0), v100, z5, tool0;
	MoveL Offs(p0,340.2,349.625, 0), v100, z5, tool0;
	MoveL Offs(p0,342.9168,350.992, 0), v100, z5, tool0;
	MoveL Offs(p0,345.5064,352.191, 0), v100, z5, tool0;
	MoveL Offs(p0,347.8176,353.14400000000006, 0), v100, z5, tool0;
	MoveL Offs(p0,349.6992,353.773, 0), v100, z5, tool0;
	MoveL Offs(p0,351.0,354.0, 0), v100, z5, tool0;
	MoveL Offs(p0,352.27040000000005,351.88160000000005, 0), v100, z5, tool0;
	MoveL Offs(p0,352.45,350.725, 0), v100, z5, tool0;
	MoveL Offs(p0,352.5696,349.33439999999996, 0), v100, z5, tool0;
	MoveL Offs(p0,352.6268,347.71819999999997, 0), v100, z5, tool0;
	MoveL Offs(p0,352.6192,345.88480000000004, 0), v100, z5, tool0;
	MoveL Offs(p0,352.54440000000005,343.8426, 0), v100, z5, tool0;
	MoveL Offs(p0,352.4,341.6, 0), v100, z5, tool0;
	MoveL Offs(p0,352.4,341.6, 0), v100, z5, tool0;
	MoveJ Offs(p0,373.6,348.8, 10), v100, z1, tool0;
	MoveL Offs(p0,376.2400000000001,348.2784000000001, 0), v100, z5, tool0;
	MoveL Offs(p0,377.4429999999999,347.9936, 0), v100, z5, tool0;
	MoveL Offs(p0,378.544,347.6992, 0), v100, z5, tool0;
	MoveL Offs(p0,379.525,347.4, 0), v100, z5, tool0;
	MoveL Offs(p0,380.368,347.1008, 0), v100, z5, tool0;
	MoveL Offs(p0,381.055,346.8064, 0), v100, z5, tool0;
	MoveL Offs(p0,381.56800000000004,346.52160000000003, 0), v100, z5, tool0;
	MoveL Offs(p0,381.889,346.25120000000004, 0), v100, z5, tool0;
	MoveL Offs(p0,382.0,346.0, 0), v100, z5, tool0;
	MoveL Offs(p0,381.22560000000004,343.36319999999995, 0), v100, z5, tool0;
	MoveL Offs(p0,380.825,342.275, 0), v100, z5, tool0;
	MoveL Offs(p0,380.35839999999996,341.0608, 0), v100, z5, tool0;
	MoveL Offs(p0,379.8342,339.7434, 0), v100, z5, tool0;
	MoveL Offs(p0,379.2608,338.3456, 0), v100, z5, tool0;
	MoveL Offs(p0,378.64660000000003,336.8902, 0), v100, z5, tool0;
	MoveL Offs(p0,378.0,335.4, 0), v100, z5, tool0;
	MoveL Offs(p0,375.76740000000007,329.61440000000005, 0), v100, z5, tool0;
	MoveL Offs(p0,374.1072000000001,323.69920000000013, 0), v100, z5, tool0;
	MoveL Offs(p0,373.01579999999996,317.71680000000003, 0), v100, z5, tool0;
	MoveL Offs(p0,372.48960000000005,311.7296, 0), v100, z5, tool0;
	MoveL Offs(p0,372.525,305.8, 0), v100, z5, tool0;
	MoveL Offs(p0,373.11839999999995,299.99039999999997, 0), v100, z5, tool0;
	MoveL Offs(p0,374.26619999999997,294.36319999999995, 0), v100, z5, tool0;
	MoveL Offs(p0,375.9648,288.9808, 0), v100, z5, tool0;
	MoveL Offs(p0,378.2106,283.9056, 0), v100, z5, tool0;
	MoveL Offs(p0,381.0,279.2, 0), v100, z5, tool0;
	MoveL Offs(p0,382.5952000000001,276.84960000000007, 0), v100, z5, tool0;
	MoveL Offs(p0,383.3148,275.74039999999997, 0), v100, z5, tool0;
	MoveL Offs(p0,383.9696,274.7008, 0), v100, z5, tool0;
	MoveL Offs(p0,384.55,273.75, 0), v100, z5, tool0;
	MoveL Offs(p0,385.0464,272.9072, 0), v100, z5, tool0;
	MoveL Offs(p0,385.4492,272.1916, 0), v100, z5, tool0;
	MoveL Offs(p0,385.7488,271.6224, 0), v100, z5, tool0;
	MoveL Offs(p0,385.9356000000001,271.2188, 0), v100, z5, tool0;
	MoveL Offs(p0,386.0,271.0, 0), v100, z5, tool0;
	MoveL Offs(p0,383.37559999999996,271.05219999999997, 0), v100, z5, tool0;
	MoveL Offs(p0,381.5072,271.8064, 0), v100, z5, tool0;
	MoveL Offs(p0,379.25,272.875, 0), v100, z5, tool0;
	MoveL Offs(p0,376.6688,274.22559999999993, 0), v100, z5, tool0;
	MoveL Offs(p0,373.8284,275.82579999999996, 0), v100, z5, tool0;
	MoveL Offs(p0,370.7936000000001,277.6432, 0), v100, z5, tool0;
	MoveL Offs(p0,367.62919999999997,279.6454, 0), v100, z5, tool0;
	MoveL Offs(p0,364.4,281.8, 0), v100, z5, tool0;
	MoveL Offs(p0,360.63880000000006,284.4698, 0), v100, z5, tool0;
	MoveL Offs(p0,356.89440000000013,287.3424000000001, 0), v100, z5, tool0;
	MoveL Offs(p0,353.3156,290.2726, 0), v100, z5, tool0;
	MoveL Offs(p0,350.0512,293.1152000000001, 0), v100, z5, tool0;
	MoveL Offs(p0,347.25,295.725, 0), v100, z5, tool0;
	MoveL Offs(p0,345.06080000000003,297.9568, 0), v100, z5, tool0;
	MoveL Offs(p0,343.6324,299.6654, 0), v100, z5, tool0;
	MoveL Offs(p0,343.1136,300.7056, 0), v100, z5, tool0;
	MoveL Offs(p0,343.6532,300.9322, 0), v100, z5, tool0;
	MoveL Offs(p0,345.4,300.2, 0), v100, z5, tool0;
	MoveL Offs(p0,347.95959999999997,299.1956, 0), v100, z5, tool0;
	MoveL Offs(p0,348.9392,298.90720000000005, 0), v100, z5, tool0;
	MoveL Offs(p0,349.95,298.65, 0), v100, z5, tool0;
	MoveL Offs(p0,350.9728,298.42879999999997, 0), v100, z5, tool0;
	MoveL Offs(p0,351.9884,298.2484, 0), v100, z5, tool0;
	MoveL Offs(p0,352.97760000000005,298.1136, 0), v100, z5, tool0;
	MoveL Offs(p0,353.9212,298.0292, 0), v100, z5, tool0;
	MoveL Offs(p0,354.8,298.0, 0), v100, z5, tool0;
	MoveL Offs(p0,357.648,298.3312000000001, 0), v100, z5, tool0;
	MoveL Offs(p0,358.616,298.8208, 0), v100, z5, tool0;
	MoveL Offs(p0,359.296,299.59360000000004, 0), v100, z5, tool0;
	MoveL Offs(p0,359.7,300.7, 0), v100, z5, tool0;
	MoveL Offs(p0,359.84000000000003,302.1904, 0), v100, z5, tool0;
	MoveL Offs(p0,359.72799999999995,304.1152, 0), v100, z5, tool0;
	MoveL Offs(p0,359.37600000000003,306.5248, 0), v100, z5, tool0;
	MoveL Offs(p0,358.796,309.4696, 0), v100, z5, tool0;
	MoveL Offs(p0,358.0,313.0, 0), v100, z5, tool0;
	MoveL Offs(p0,357.0520000000001,317.11480000000006, 0), v100, z5, tool0;
	MoveL Offs(p0,356.2480000000001,321.0544000000001, 0), v100, z5, tool0;
	MoveL Offs(p0,355.58799999999997,324.81160000000006, 0), v100, z5, tool0;
	MoveL Offs(p0,355.072,328.3792, 0), v100, z5, tool0;
	MoveL Offs(p0,354.7,331.75, 0), v100, z5, tool0;
	MoveL Offs(p0,354.4719999999999,334.91679999999997, 0), v100, z5, tool0;
	MoveL Offs(p0,354.38800000000003,337.87239999999997, 0), v100, z5, tool0;
	MoveL Offs(p0,354.44800000000004,340.60960000000006, 0), v100, z5, tool0;
	MoveL Offs(p0,354.65200000000004,343.12120000000004, 0), v100, z5, tool0;
	MoveL Offs(p0,355.0,345.4, 0), v100, z5, tool0;
	MoveL Offs(p0,355.6016000000001,348.4032000000001, 0), v100, z5, tool0;
	MoveL Offs(p0,355.9324,349.4878, 0), v100, z5, tool0;
	MoveL Offs(p0,356.3088,350.32160000000005, 0), v100, z5, tool0;
	MoveL Offs(p0,356.75,350.925, 0), v100, z5, tool0;
	MoveL Offs(p0,357.27520000000004,351.3184, 0), v100, z5, tool0;
	MoveL Offs(p0,357.9036,351.5222, 0), v100, z5, tool0;
	MoveL Offs(p0,358.6544,351.5568, 0), v100, z5, tool0;
	MoveL Offs(p0,359.5468,351.4426, 0), v100, z5, tool0;
	MoveL Offs(p0,360.6,351.2, 0), v100, z5, tool0;
	MoveL Offs(p0,363.5592,350.4422, 0), v100, z5, tool0;
	MoveL Offs(p0,364.83040000000005,350.1824, 0), v100, z5, tool0;
	MoveL Offs(p0,366.2,349.925, 0), v100, z5, tool0;
	MoveL Offs(p0,367.64160000000004,349.67359999999996, 0), v100, z5, tool0;
	MoveL Offs(p0,369.1288,349.4318, 0), v100, z5, tool0;
	MoveL Offs(p0,370.63520000000005,349.20320000000004, 0), v100, z5, tool0;
	MoveL Offs(p0,372.1344,348.9914, 0), v100, z5, tool0;
	MoveL Offs(p0,373.6,348.8, 0), v100, z5, tool0;
	MoveL Offs(p0,373.6,348.8, 0), v100, z5, tool0;
	MoveJ Offs(p0,328.6,328.6, 10), v100, z1, tool0;
	MoveL Offs(p0,329.04640000000006,326.0912000000001, 0), v100, z5, tool0;
	MoveL Offs(p0,329.1436,325.28079999999994, 0), v100, z5, tool0;
	MoveL Offs(p0,329.1472,324.75360000000006, 0), v100, z5, tool0;
	MoveL Offs(p0,329.05,324.5, 0), v100, z5, tool0;
	MoveL Offs(p0,328.84479999999996,324.5104, 0), v100, z5, tool0;
	MoveL Offs(p0,328.52439999999996,324.77520000000004, 0), v100, z5, tool0;
	MoveL Offs(p0,328.08160000000004,325.2848, 0), v100, z5, tool0;
	MoveL Offs(p0,327.5092,326.0296, 0), v100, z5, tool0;
	MoveL Offs(p0,325.27520000000004,329.61920000000003, 0), v100, z5, tool0;
	MoveL Offs(p0,324.73179999999996,330.9258, 0), v100, z5, tool0;
	MoveL Offs(p0,324.34560000000005,332.1616000000001, 0), v100, z5, tool0;
	MoveL Offs(p0,324.125,333.275, 0), v100, z5, tool0;
	MoveL Offs(p0,324.0784,334.21439999999996, 0), v100, z5, tool0;
	MoveL Offs(p0,324.2142,334.9282, 0), v100, z5, tool0;
	MoveL Offs(p0,324.54080000000005,335.3648, 0), v100, z5, tool0;
	MoveL Offs(p0,325.0666,335.4726, 0), v100, z5, tool0;
	MoveL Offs(p0,325.8,335.2, 0), v100, z5, tool0;
	MoveL Offs(p0,327.35,332.8, 0), v100, z5, tool0;
	MoveL Offs(p0,327.64320000000004,332.0464, 0), v100, z5, tool0;
	MoveL Offs(p0,327.9196,331.23519999999996, 0), v100, z5, tool0;
	MoveL Offs(p0,328.17440000000005,330.3808, 0), v100, z5, tool0;
	MoveL Offs(p0,328.40279999999996,329.49760000000003, 0), v100, z5, tool0;
	MoveL Offs(p0,328.6,328.6, 0), v100, z5, tool0;
	MoveL Offs(p0,328.6,328.6, 0), v100, z5, tool0;
	MoveJ Offs(p0,57.0,327.6, 10), v100, z1, tool0;
	MoveL Offs(p0,56.2752,324.47740000000005, 0), v100, z5, tool0;
	MoveL Offs(p0,55.665600000000026,320.4272000000001, 0), v100, z5, tool0;
	MoveL Offs(p0,55.178399999999996,315.6858, 0), v100, z5, tool0;
	MoveL Offs(p0,54.820800000000006,310.4896, 0), v100, z5, tool0;
	MoveL Offs(p0,54.6,305.075, 0), v100, z5, tool0;
	MoveL Offs(p0,54.523199999999996,299.67839999999995, 0), v100, z5, tool0;
	MoveL Offs(p0,54.5976,294.5362, 0), v100, z5, tool0;
	MoveL Offs(p0,54.83040000000001,289.8848, 0), v100, z5, tool0;
	MoveL Offs(p0,55.2288,285.9606, 0), v100, z5, tool0;
	MoveL Offs(p0,55.8,283.0, 0), v100, z5, tool0;
	MoveL Offs(p0,56.44640000000002,280.38560000000007, 0), v100, z5, tool0;
	MoveL Offs(p0,56.712599999999995,279.1264, 0), v100, z5, tool0;
	MoveL Offs(p0,56.93920000000001,277.92480000000006, 0), v100, z5, tool0;
	MoveL Offs(p0,57.125,276.8, 0), v100, z5, tool0;
	MoveL Offs(p0,57.2688,275.7712, 0), v100, z5, tool0;
	MoveL Offs(p0,57.3694,274.8576, 0), v100, z5, tool0;
	MoveL Offs(p0,57.42560000000001,274.07840000000004, 0), v100, z5, tool0;
	MoveL Offs(p0,57.4362,273.4528, 0), v100, z5, tool0;
	MoveL Offs(p0,57.4,273.0, 0), v100, z5, tool0;
	MoveL Offs(p0,54.5,270.7, 0), v100, z5, tool0;
	MoveL Offs(p0,53.411199999999994,270.12, 0), v100, z5, tool0;
	MoveL Offs(p0,52.19759999999999,269.52799999999996, 0), v100, z5, tool0;
	MoveL Offs(p0,50.878400000000006,268.93600000000004, 0), v100, z5, tool0;
	MoveL Offs(p0,49.47280000000001,268.356, 0), v100, z5, tool0;
	MoveL Offs(p0,48.0,267.8, 0), v100, z5, tool0;
	MoveL Offs(p0,44.98560000000001,266.7072000000001, 0), v100, z5, tool0;
	MoveL Offs(p0,43.5054,266.1637999999999, 0), v100, z5, tool0;
	MoveL Offs(p0,42.076800000000006,265.6336, 0), v100, z5, tool0;
	MoveL Offs(p0,40.725,265.125, 0), v100, z5, tool0;
	MoveL Offs(p0,39.4752,264.64639999999997, 0), v100, z5, tool0;
	MoveL Offs(p0,38.352599999999995,264.20619999999997, 0), v100, z5, tool0;
	MoveL Offs(p0,37.382400000000004,263.81280000000004, 0), v100, z5, tool0;
	MoveL Offs(p0,36.589800000000004,263.4746, 0), v100, z5, tool0;
	MoveL Offs(p0,36.0,263.2, 0), v100, z5, tool0;
	MoveL Offs(p0,33.4688,264.0416, 0), v100, z5, tool0;
	MoveL Offs(p0,32.95,265.05, 0), v100, z5, tool0;
	MoveL Offs(p0,32.4432,266.45439999999996, 0), v100, z5, tool0;
	MoveL Offs(p0,31.931599999999996,268.29319999999996, 0), v100, z5, tool0;
	MoveL Offs(p0,31.398400000000002,270.6048, 0), v100, z5, tool0;
	MoveL Offs(p0,30.826800000000002,273.42760000000004, 0), v100, z5, tool0;
	MoveL Offs(p0,30.2,276.8, 0), v100, z5, tool0;
	MoveL Offs(p0,29.296000000000003,281.74080000000004, 0), v100, z5, tool0;
	MoveL Offs(p0,28.272000000000002,286.1104000000001, 0), v100, z5, tool0;
	MoveL Offs(p0,27.139999999999997,289.8896, 0), v100, z5, tool0;
	MoveL Offs(p0,25.912,293.05920000000003, 0), v100, z5, tool0;
	MoveL Offs(p0,24.6,295.6, 0), v100, z5, tool0;
	MoveL Offs(p0,23.216,297.4928, 0), v100, z5, tool0;
	MoveL Offs(p0,21.772,298.71840000000003, 0), v100, z5, tool0;
	MoveL Offs(p0,20.28,299.2576, 0), v100, z5, tool0;
	MoveL Offs(p0,18.752000000000002,299.0912, 0), v100, z5, tool0;
	MoveL Offs(p0,17.2,298.2, 0), v100, z5, tool0;
	MoveL Offs(p0,15.4666,296.0814, 0), v100, z5, tool0;
	MoveL Offs(p0,14.8672,295.06080000000003, 0), v100, z5, tool0;
	MoveL Offs(p0,14.275,293.925, 0), v100, z5, tool0;
	MoveL Offs(p0,13.700799999999997,292.6992, 0), v100, z5, tool0;
	MoveL Offs(p0,13.1554,291.4086, 0), v100, z5, tool0;
	MoveL Offs(p0,12.649600000000001,290.0784, 0), v100, z5, tool0;
	MoveL Offs(p0,12.1942,288.73380000000003, 0), v100, z5, tool0;
	MoveL Offs(p0,11.8,287.4, 0), v100, z5, tool0;
	MoveL Offs(p0,11.075000000000001,283.956, 0), v100, z5, tool0;
	MoveL Offs(p0,10.464000000000002,279.648, 0), v100, z5, tool0;
	MoveL Offs(p0,9.973,274.692, 0), v100, z5, tool0;
	MoveL Offs(p0,9.608,269.304, 0), v100, z5, tool0;
	MoveL Offs(p0,9.375,263.7, 0), v100, z5, tool0;
	MoveL Offs(p0,9.28,258.09599999999995, 0), v100, z5, tool0;
	MoveL Offs(p0,9.328999999999999,252.708, 0), v100, z5, tool0;
	MoveL Offs(p0,9.528,247.752, 0), v100, z5, tool0;
	MoveL Offs(p0,9.883,243.44400000000002, 0), v100, z5, tool0;
	MoveL Offs(p0,10.4,240.0, 0), v100, z5, tool0;
	MoveL Offs(p0,11.044800000000002,237.05760000000004, 0), v100, z5, tool0;
	MoveL Offs(p0,11.2172,236.0634, 0), v100, z5, tool0;
	MoveL Offs(p0,11.2864,235.3728, 0), v100, z5, tool0;
	MoveL Offs(p0,11.25,234.975, 0), v100, z5, tool0;
	MoveL Offs(p0,11.105599999999999,234.85920000000002, 0), v100, z5, tool0;
	MoveL Offs(p0,10.8508,235.01459999999997, 0), v100, z5, tool0;
	MoveL Offs(p0,10.483200000000002,235.43040000000002, 0), v100, z5, tool0;
	MoveL Offs(p0,10.0004,236.0958, 0), v100, z5, tool0;
	MoveL Offs(p0,9.4,237.0, 0), v100, z5, tool0;
	MoveL Offs(p0,8.536000000000003,239.38560000000007, 0), v100, z5, tool0;
	MoveL Offs(p0,8.175999999999998,241.1814, 0), v100, z5, tool0;
	MoveL Offs(p0,7.864,243.3648, 0), v100, z5, tool0;
	MoveL Offs(p0,7.6,245.925, 0), v100, z5, tool0;
	MoveL Offs(p0,7.383999999999999,248.85119999999998, 0), v100, z5, tool0;
	MoveL Offs(p0,7.215999999999999,252.1326, 0), v100, z5, tool0;
	MoveL Offs(p0,7.096000000000001,255.75840000000002, 0), v100, z5, tool0;
	MoveL Offs(p0,7.024000000000001,259.7178, 0), v100, z5, tool0;
	MoveL Offs(p0,7.0,264.0, 0), v100, z5, tool0;
	MoveL Offs(p0,7.094800000000001,271.32460000000003, 0), v100, z5, tool0;
	MoveL Offs(p0,7.398400000000002,277.8848000000001, 0), v100, z5, tool0;
	MoveL Offs(p0,7.9396,283.7802, 0), v100, z5, tool0;
	MoveL Offs(p0,8.7472,289.1104, 0), v100, z5, tool0;
	MoveL Offs(p0,9.85,293.975, 0), v100, z5, tool0;
	MoveL Offs(p0,11.276800000000001,298.4736, 0), v100, z5, tool0;
	MoveL Offs(p0,13.056400000000002,302.7058, 0), v100, z5, tool0;
	MoveL Offs(p0,15.217600000000001,306.7712, 0), v100, z5, tool0;
	MoveL Offs(p0,17.7892,310.7694, 0), v100, z5, tool0;
	MoveL Offs(p0,20.8,314.8, 0), v100, z5, tool0;
	MoveL Offs(p0,23.1,317.32280000000003, 0), v100, z5, tool0;
	MoveL Offs(p0,25.856000000000012,319.8144000000001, 0), v100, z5, tool0;
	MoveL Offs(p0,28.972,322.21959999999996, 0), v100, z5, tool0;
	MoveL Offs(p0,32.35200000000001,324.4832, 0), v100, z5, tool0;
	MoveL Offs(p0,35.9,326.55, 0), v100, z5, tool0;
	MoveL Offs(p0,39.52,328.36479999999995, 0), v100, z5, tool0;
	MoveL Offs(p0,43.116,329.8724, 0), v100, z5, tool0;
	MoveL Offs(p0,46.592000000000006,331.0176, 0), v100, z5, tool0;
	MoveL Offs(p0,49.852,331.7452, 0), v100, z5, tool0;
	MoveL Offs(p0,52.8,332.0, 0), v100, z5, tool0;
	MoveL Offs(p0,55.272000000000006,331.9072000000001, 0), v100, z5, tool0;
	MoveL Offs(p0,56.138999999999996,331.7678, 0), v100, z5, tool0;
	MoveL Offs(p0,56.784000000000006,331.54560000000004, 0), v100, z5, tool0;
	MoveL Offs(p0,57.225,331.225, 0), v100, z5, tool0;
	MoveL Offs(p0,57.48,330.7904, 0), v100, z5, tool0;
	MoveL Offs(p0,57.56699999999999,330.22619999999995, 0), v100, z5, tool0;
	MoveL Offs(p0,57.504000000000005,329.5168, 0), v100, z5, tool0;
	MoveL Offs(p0,57.309000000000005,328.6466, 0), v100, z5, tool0;
	MoveL Offs(p0,57.0,327.6, 0), v100, z5, tool0;
	MoveL Offs(p0,57.0,327.6, 0), v100, z5, tool0;
	MoveJ Offs(p0,156.0,315.6, 10), v100, z1, tool0;
	MoveL Offs(p0,155.7366,309.921, 0), v100, z5, tool0;
	MoveL Offs(p0,154.99680000000004,302.5200000000001, 0), v100, z5, tool0;
	MoveL Offs(p0,153.8562,293.811, 0), v100, z5, tool0;
	MoveL Offs(p0,152.39040000000003,284.208, 0), v100, z5, tool0;
	MoveL Offs(p0,150.675,274.125, 0), v100, z5, tool0;
	MoveL Offs(p0,148.7856,263.976, 0), v100, z5, tool0;
	MoveL Offs(p0,146.7978,254.175, 0), v100, z5, tool0;
	MoveL Offs(p0,144.7872,245.13600000000002, 0), v100, z5, tool0;
	MoveL Offs(p0,142.8294,237.273, 0), v100, z5, tool0;
	MoveL Offs(p0,141.0,231.0, 0), v100, z5, tool0;
	MoveL Offs(p0,143.8574,234.171, 0), v100, z5, tool0;
	MoveL Offs(p0,144.86560000000003,235.704, 0), v100, z5, tool0;
	MoveL Offs(p0,145.98420000000002,237.45300000000003, 0), v100, z5, tool0;
	MoveL Offs(p0,147.2,239.4, 0), v100, z5, tool0;
	MoveL Offs(p0,149.92400000000004,243.6538, 0), v100, z5, tool0;
	MoveL Offs(p0,152.21600000000007,246.81440000000012, 0), v100, z5, tool0;
	MoveL Offs(p0,154.07599999999996,248.88060000000002, 0), v100, z5, tool0;
	MoveL Offs(p0,155.50400000000002,249.8512, 0), v100, z5, tool0;
	MoveL Offs(p0,156.5,249.725, 0), v100, z5, tool0;
	MoveL Offs(p0,157.064,248.50079999999997, 0), v100, z5, tool0;
	MoveL Offs(p0,157.196,246.17739999999998, 0), v100, z5, tool0;
	MoveL Offs(p0,156.89600000000002,242.7536, 0), v100, z5, tool0;
	MoveL Offs(p0,156.164,238.22820000000002, 0), v100, z5, tool0;
	MoveL Offs(p0,155.0,232.6, 0), v100, z5, tool0;
	MoveL Offs(p0,153.489,226.25120000000007, 0), v100, z5, tool0;
	MoveL Offs(p0,151.74400000000006,219.87360000000007, 0), v100, z5, tool0;
	MoveL Offs(p0,149.80699999999996,213.57039999999998, 0), v100, z5, tool0;
	MoveL Offs(p0,147.72000000000003,207.44480000000004, 0), v100, z5, tool0;
	MoveL Offs(p0,145.525,201.6, 0), v100, z5, tool0;
	MoveL Offs(p0,143.26399999999998,196.13920000000002, 0), v100, z5, tool0;
	MoveL Offs(p0,140.97899999999998,191.16559999999998, 0), v100, z5, tool0;
	MoveL Offs(p0,138.71200000000002,186.7824, 0), v100, z5, tool0;
	MoveL Offs(p0,136.505,183.0928, 0), v100, z5, tool0;
	MoveL Offs(p0,134.4,180.2, 0), v100, z5, tool0;
	MoveL Offs(p0,128.8,173.4, 0), v100, z5, tool0;
	MoveL Offs(p0,122.4,184.4, 0), v100, z5, tool0;
	MoveL Offs(p0,119.9728,188.53600000000006, 0), v100, z5, tool0;
	MoveL Offs(p0,118.5192,190.84400000000002, 0), v100, z5, tool0;
	MoveL Offs(p0,116.95039999999999,193.248, 0), v100, z5, tool0;
	MoveL Offs(p0,115.3,195.7, 0), v100, z5, tool0;
	MoveL Offs(p0,113.6016,198.152, 0), v100, z5, tool0;
	MoveL Offs(p0,111.88879999999999,200.55599999999998, 0), v100, z5, tool0;
	MoveL Offs(p0,110.19520000000003,202.864, 0), v100, z5, tool0;
	MoveL Offs(p0,108.55440000000002,205.02800000000002, 0), v100, z5, tool0;
	MoveL Offs(p0,107.0,207.0, 0), v100, z5, tool0;
	MoveL Offs(p0,97.6,218.4, 0), v100, z5, tool0;
	MoveL Offs(p0,101.8,233.6, 0), v100, z5, tool0;
	MoveL Offs(p0,102.4642,236.31380000000004, 0), v100, z5, tool0;
	MoveL Offs(p0,103.12960000000002,239.25440000000012, 0), v100, z5, tool0;
	MoveL Offs(p0,103.78539999999998,242.36060000000003, 0), v100, z5, tool0;
	MoveL Offs(p0,104.42080000000001,245.57120000000003, 0), v100, z5, tool0;
	MoveL Offs(p0,105.025,248.825, 0), v100, z5, tool0;
	MoveL Offs(p0,105.58720000000001,252.06080000000003, 0), v100, z5, tool0;
	MoveL Offs(p0,106.0966,255.2174, 0), v100, z5, tool0;
	MoveL Offs(p0,106.5424,258.2336, 0), v100, z5, tool0;
	MoveL Offs(p0,106.9138,261.0482, 0), v100, z5, tool0;
	MoveL Offs(p0,107.2,263.6, 0), v100, z5, tool0;
	MoveL Offs(p0,107.4514,265.89860000000004, 0), v100, z5, tool0;
	MoveL Offs(p0,107.72320000000005,268.09280000000007, 0), v100, z5, tool0;
	MoveL Offs(p0,108.0118,270.1502, 0), v100, z5, tool0;
	MoveL Offs(p0,108.31360000000002,272.0384, 0), v100, z5, tool0;
	MoveL Offs(p0,108.625,273.725, 0), v100, z5, tool0;
	MoveL Offs(p0,108.94239999999999,275.1776, 0), v100, z5, tool0;
	MoveL Offs(p0,109.2622,276.36379999999997, 0), v100, z5, tool0;
	MoveL Offs(p0,109.5808,277.25120000000004, 0), v100, z5, tool0;
	MoveL Offs(p0,109.8946,277.80740000000003, 0), v100, z5, tool0;
	MoveL Offs(p0,110.2,278.0, 0), v100, z5, tool0;
	MoveL Offs(p0,112.68640000000002,274.67199999999997, 0), v100, z5, tool0;
	MoveL Offs(p0,113.2,273.0, 0), v100, z5, tool0;
	MoveL Offs(p0,113.6416,271.088, 0), v100, z5, tool0;
	MoveL Offs(p0,113.99680000000001,268.98400000000004, 0), v100, z5, tool0;
	MoveL Offs(p0,114.25120000000001,266.736, 0), v100, z5, tool0;
	MoveL Offs(p0,114.3904,264.392, 0), v100, z5, tool0;
	MoveL Offs(p0,114.4,262.0, 0), v100, z5, tool0;
	MoveL Offs(p0,114.35680000000005,259.1312000000001, 0), v100, z5, tool0;
	MoveL Offs(p0,114.3982,258.1408, 0), v100, z5, tool0;
	MoveL Offs(p0,114.4864,257.4336, 0), v100, z5, tool0;
	MoveL Offs(p0,114.625,257.0, 0), v100, z5, tool0;
	MoveL Offs(p0,114.8176,256.8304, 0), v100, z5, tool0;
	MoveL Offs(p0,115.06779999999999,256.91519999999997, 0), v100, z5, tool0;
	MoveL Offs(p0,115.37920000000001,257.24480000000005, 0), v100, z5, tool0;
	MoveL Offs(p0,115.75540000000001,257.8096, 0), v100, z5, tool0;
	MoveL Offs(p0,116.2,258.6, 0), v100, z5, tool0;
	MoveL Offs(p0,117.00460000000001,260.7798, 0), v100, z5, tool0;
	MoveL Offs(p0,117.83680000000007,264.56640000000004, 0), v100, z5, tool0;
	MoveL Offs(p0,118.66420000000001,269.61060000000003, 0), v100, z5, tool0;
	MoveL Offs(p0,119.4544,275.56319999999994, 0), v100, z5, tool0;
	MoveL Offs(p0,120.175,282.075, 0), v100, z5, tool0;
	MoveL Offs(p0,120.7936,288.79679999999996, 0), v100, z5, tool0;
	MoveL Offs(p0,121.27779999999998,295.37940000000003, 0), v100, z5, tool0;
	MoveL Offs(p0,121.59520000000002,301.4736, 0), v100, z5, tool0;
	MoveL Offs(p0,121.71340000000001,306.7302, 0), v100, z5, tool0;
	MoveL Offs(p0,121.6,310.8, 0), v100, z5, tool0;
	MoveL Offs(p0,121.49760000000003,313.3456000000001, 0), v100, z5, tool0;
	MoveL Offs(p0,121.5424,314.52239999999995, 0), v100, z5, tool0;
	MoveL Offs(p0,121.64479999999999,315.61280000000005, 0), v100, z5, tool0;
	MoveL Offs(p0,121.8,316.6, 0), v100, z5, tool0;
	MoveL Offs(p0,122.00319999999999,317.4672, 0), v100, z5, tool0;
	MoveL Offs(p0,122.24959999999999,318.1976, 0), v100, z5, tool0;
	MoveL Offs(p0,122.5344,318.77440000000007, 0), v100, z5, tool0;
	MoveL Offs(p0,122.85280000000003,319.1808, 0), v100, z5, tool0;
	MoveL Offs(p0,123.2,319.4, 0), v100, z5, tool0;
	MoveL Offs(p0,125.60000000000005,317.4992000000001, 0), v100, z5, tool0;
	MoveL Offs(p0,127.025,315.0458, 0), v100, z5, tool0;
	MoveL Offs(p0,128.48,311.9216, 0), v100, z5, tool0;
	MoveL Offs(p0,129.875,308.375, 0), v100, z5, tool0;
	MoveL Offs(p0,131.12,304.6544, 0), v100, z5, tool0;
	MoveL Offs(p0,132.125,301.0082, 0), v100, z5, tool0;
	MoveL Offs(p0,132.8,297.68480000000005, 0), v100, z5, tool0;
	MoveL Offs(p0,133.055,294.9326, 0), v100, z5, tool0;
	MoveL Offs(p0,132.8,293.0, 0), v100, z5, tool0;
	MoveL Offs(p0,132.325,290.725, 0), v100, z5, tool0;
	MoveL Offs(p0,132.3968,290.48, 0), v100, z5, tool0;
	MoveL Offs(p0,132.5214,290.319, 0), v100, z5, tool0;
	MoveL Offs(p0,132.69760000000002,290.24800000000005, 0), v100, z5, tool0;
	MoveL Offs(p0,132.9242,290.273, 0), v100, z5, tool0;
	MoveL Offs(p0,133.2,290.4, 0), v100, z5, tool0;
	MoveL Offs(p0,134.92620000000002,292.848, 0), v100, z5, tool0;
	MoveL Offs(p0,135.8144,294.33600000000007, 0), v100, z5, tool0;
	MoveL Offs(p0,136.825,296.1, 0), v100, z5, tool0;
	MoveL Offs(p0,137.9376,298.10400000000004, 0), v100, z5, tool0;
	MoveL Offs(p0,139.1318,300.312, 0), v100, z5, tool0;
	MoveL Offs(p0,140.38720000000004,302.688, 0), v100, z5, tool0;
	MoveL Offs(p0,141.68339999999998,305.196, 0), v100, z5, tool0;
	MoveL Offs(p0,143.0,307.8, 0), v100, z5, tool0;
	MoveL Offs(p0,145.50240000000002,312.79200000000003, 0), v100, z5, tool0;
	MoveL Offs(p0,147.73120000000003,316.84800000000007, 0), v100, z5, tool0;
	MoveL Offs(p0,149.68880000000001,319.96799999999996, 0), v100, z5, tool0;
	MoveL Offs(p0,151.37759999999997,322.152, 0), v100, z5, tool0;
	MoveL Offs(p0,152.8,323.4, 0), v100, z5, tool0;
	MoveL Offs(p0,153.95839999999998,323.712, 0), v100, z5, tool0;
	MoveL Offs(p0,154.85520000000002,323.088, 0), v100, z5, tool0;
	MoveL Offs(p0,155.4928,321.528, 0), v100, z5, tool0;
	MoveL Offs(p0,155.8736,319.03200000000004, 0), v100, z5, tool0;
	MoveL Offs(p0,156.0,315.6, 0), v100, z5, tool0;
	MoveL Offs(p0,156.0,315.6, 0), v100, z5, tool0;
	MoveJ Offs(p0,94.6,283.4, 10), v100, z1, tool0;
	MoveL Offs(p0,94.64260000000003,281.26900000000006, 0), v100, z5, tool0;
	MoveL Offs(p0,94.65280000000003,279.2160000000001, 0), v100, z5, tool0;
	MoveL Offs(p0,94.63419999999999,277.271, 0), v100, z5, tool0;
	MoveL Offs(p0,94.59040000000002,275.464, 0), v100, z5, tool0;
	MoveL Offs(p0,94.525,273.825, 0), v100, z5, tool0;
	MoveL Offs(p0,94.44160000000001,272.38399999999996, 0), v100, z5, tool0;
	MoveL Offs(p0,94.3438,271.171, 0), v100, z5, tool0;
	MoveL Offs(p0,94.2352,270.216, 0), v100, z5, tool0;
	MoveL Offs(p0,94.11940000000001,269.54900000000004, 0), v100, z5, tool0;
	MoveL Offs(p0,94.0,269.2, 0), v100, z5, tool0;
	MoveL Offs(p0,91.424,269.1008, 0), v100, z5, tool0;
	MoveL Offs(p0,90.3,269.25, 0), v100, z5, tool0;
	MoveL Offs(p0,89.032,269.4592, 0), v100, z5, tool0;
	MoveL Offs(p0,87.64399999999999,269.7236, 0), v100, z5, tool0;
	MoveL Offs(p0,86.16000000000001,270.0384, 0), v100, z5, tool0;
	MoveL Offs(p0,84.604,270.39880000000005, 0), v100, z5, tool0;
	MoveL Offs(p0,83.0,270.8, 0), v100, z5, tool0;
	MoveL Offs(p0,80.45100000000001,271.4102000000001, 0), v100, z5, tool0;
	MoveL Offs(p0,78.42400000000002,271.9376000000001, 0), v100, z5, tool0;
	MoveL Offs(p0,76.889,272.4074, 0), v100, z5, tool0;
	MoveL Offs(p0,75.816,272.8448, 0), v100, z5, tool0;
	MoveL Offs(p0,75.175,273.275, 0), v100, z5, tool0;
	MoveL Offs(p0,74.936,273.7232, 0), v100, z5, tool0;
	MoveL Offs(p0,75.069,274.21459999999996, 0), v100, z5, tool0;
	MoveL Offs(p0,75.54400000000001,274.7744, 0), v100, z5, tool0;
	MoveL Offs(p0,76.331,275.42780000000005, 0), v100, z5, tool0;
	MoveL Offs(p0,77.4,276.2, 0), v100, z5, tool0;
	MoveL Offs(p0,80.70720000000003,279.2464000000001, 0), v100, z5, tool0;
	MoveL Offs(p0,82.41479999999999,281.2976, 0), v100, z5, tool0;
	MoveL Offs(p0,84.08160000000001,283.5792, 0), v100, z5, tool0;
	MoveL Offs(p0,85.65,286.0, 0), v100, z5, tool0;
	MoveL Offs(p0,87.0624,288.4688, 0), v100, z5, tool0;
	MoveL Offs(p0,88.2612,290.8944, 0), v100, z5, tool0;
	MoveL Offs(p0,89.18880000000001,293.1856, 0), v100, z5, tool0;
	MoveL Offs(p0,89.78760000000001,295.25120000000004, 0), v100, z5, tool0;
	MoveL Offs(p0,90.0,297.0, 0), v100, z5, tool0;
	MoveL Offs(p0,90.30080000000001,299.15999999999997, 0), v100, z5, tool0;
	MoveL Offs(p0,90.475,299.4, 0), v100, z5, tool0;
	MoveL Offs(p0,90.69120000000001,299.52, 0), v100, z5, tool0;
	MoveL Offs(p0,90.9506,299.52, 0), v100, z5, tool0;
	MoveL Offs(p0,91.2544,299.4, 0), v100, z5, tool0;
	MoveL Offs(p0,91.6038,299.16, 0), v100, z5, tool0;
	MoveL Offs(p0,92.0,298.8, 0), v100, z5, tool0;
	MoveL Offs(p0,93.053,296.34299999999996, 0), v100, z5, tool0;
	MoveL Offs(p0,93.376,294.992, 0), v100, z5, tool0;
	MoveL Offs(p0,93.675,293.425, 0), v100, z5, tool0;
	MoveL Offs(p0,93.94399999999999,291.672, 0), v100, z5, tool0;
	MoveL Offs(p0,94.17699999999999,289.76300000000003, 0), v100, z5, tool0;
	MoveL Offs(p0,94.36800000000001,287.728, 0), v100, z5, tool0;
	MoveL Offs(p0,94.51100000000001,285.59700000000004, 0), v100, z5, tool0;
	MoveL Offs(p0,94.6,283.4, 0), v100, z5, tool0;
	MoveL Offs(p0,94.6,283.4, 0), v100, z5, tool0;
	MoveJ Offs(p0,23.6,292.6, 10), v100, z1, tool0;
	MoveL Offs(p0,24.814999999999998,289.29879999999997, 0), v100, z5, tool0;
	MoveL Offs(p0,25.264000000000003,287.6336, 0), v100, z5, tool0;
	MoveL Offs(p0,25.725,285.75, 0), v100, z5, tool0;
	MoveL Offs(p0,26.191999999999997,283.6864, 0), v100, z5, tool0;
	MoveL Offs(p0,26.659,281.4812, 0), v100, z5, tool0;
	MoveL Offs(p0,27.120000000000005,279.1728, 0), v100, z5, tool0;
	MoveL Offs(p0,27.569000000000006,276.7996, 0), v100, z5, tool0;
	MoveL Offs(p0,28.0,274.4, 0), v100, z5, tool0;
	MoveL Offs(p0,28.6456,270.48120000000006, 0), v100, z5, tool0;
	MoveL Offs(p0,29.13280000000001,267.2896, 0), v100, z5, tool0;
	MoveL Offs(p0,29.4472,264.7124, 0), v100, z5, tool0;
	MoveL Offs(p0,29.574400000000004,262.63680000000005, 0), v100, z5, tool0;
	MoveL Offs(p0,29.5,260.95, 0), v100, z5, tool0;
	MoveL Offs(p0,29.209600000000002,259.5392, 0), v100, z5, tool0;
	MoveL Offs(p0,28.688799999999997,258.29159999999996, 0), v100, z5, tool0;
	MoveL Offs(p0,27.9232,257.09440000000006, 0), v100, z5, tool0;
	MoveL Offs(p0,26.898400000000002,255.8348, 0), v100, z5, tool0;
	MoveL Offs(p0,25.6,254.4, 0), v100, z5, tool0;
	MoveL Offs(p0,22.9342,251.36520000000002, 0), v100, z5, tool0;
	MoveL Offs(p0,22.0224,250.2624, 0), v100, z5, tool0;
	MoveL Offs(p0,21.125,249.15, 0), v100, z5, tool0;
	MoveL Offs(p0,20.257599999999996,248.0496, 0), v100, z5, tool0;
	MoveL Offs(p0,19.4358,246.9828, 0), v100, z5, tool0;
	MoveL Offs(p0,18.6752,245.97120000000004, 0), v100, z5, tool0;
	MoveL Offs(p0,17.991400000000002,245.03640000000001, 0), v100, z5, tool0;
	MoveL Offs(p0,17.4,244.2, 0), v100, z5, tool0;
	MoveL Offs(p0,14.2,239.4, 0), v100, z5, tool0;
	MoveL Offs(p0,12.8,244.8, 0), v100, z5, tool0;
	MoveL Offs(p0,12.316800000000002,247.91400000000007, 0), v100, z5, tool0;
	MoveL Offs(p0,12.054400000000005,252.24000000000007, 0), v100, z5, tool0;
	MoveL Offs(p0,11.993599999999999,257.454, 0), v100, z5, tool0;
	MoveL Offs(p0,12.115200000000002,263.232, 0), v100, z5, tool0;
	MoveL Offs(p0,12.4,269.25, 0), v100, z5, tool0;
	MoveL Offs(p0,12.828800000000001,275.184, 0), v100, z5, tool0;
	MoveL Offs(p0,13.3824,280.71, 0), v100, z5, tool0;
	MoveL Offs(p0,14.041599999999999,285.504, 0), v100, z5, tool0;
	MoveL Offs(p0,14.787200000000002,289.242, 0), v100, z5, tool0;
	MoveL Offs(p0,15.6,291.6, 0), v100, z5, tool0;
	MoveL Offs(p0,17.353600000000007,294.21920000000006, 0), v100, z5, tool0;
	MoveL Offs(p0,18.197400000000002,295.06679999999994, 0), v100, z5, tool0;
	MoveL Offs(p0,19.0208,295.60960000000006, 0), v100, z5, tool0;
	MoveL Offs(p0,19.825,295.85, 0), v100, z5, tool0;
	MoveL Offs(p0,20.6112,295.79040000000003, 0), v100, z5, tool0;
	MoveL Offs(p0,21.380599999999998,295.4332, 0), v100, z5, tool0;
	MoveL Offs(p0,22.1344,294.7808, 0), v100, z5, tool0;
	MoveL Offs(p0,22.8738,293.8356, 0), v100, z5, tool0;
	MoveL Offs(p0,23.6,292.6, 0), v100, z5, tool0;
	MoveL Offs(p0,23.6,292.6, 0), v100, z5, tool0;
	MoveJ Offs(p0,346.6,267.4, 10), v100, z1, tool0;
	MoveL Offs(p0,346.3968000000001,262.95660000000004, 0), v100, z5, tool0;
	MoveL Offs(p0,346.27040000000005,258.9488000000001, 0), v100, z5, tool0;
	MoveL Offs(p0,346.2256,255.32020000000003, 0), v100, z5, tool0;
	MoveL Offs(p0,346.26720000000006,252.01440000000002, 0), v100, z5, tool0;
	MoveL Offs(p0,346.4,248.975, 0), v100, z5, tool0;
	MoveL Offs(p0,346.62880000000007,246.1456, 0), v100, z5, tool0;
	MoveL Offs(p0,346.9584,243.46980000000002, 0), v100, z5, tool0;
	MoveL Offs(p0,347.39360000000005,240.89120000000003, 0), v100, z5, tool0;
	MoveL Offs(p0,347.9392,238.35340000000002, 0), v100, z5, tool0;
	MoveL Offs(p0,348.6,235.8, 0), v100, z5, tool0;
	MoveL Offs(p0,349.91760000000005,231.7772, 0), v100, z5, tool0;
	MoveL Offs(p0,351.3408000000001,228.1216000000001, 0), v100, z5, tool0;
	MoveL Offs(p0,352.85519999999997,224.8524, 0), v100, z5, tool0;
	MoveL Offs(p0,354.44640000000004,221.98880000000003, 0), v100, z5, tool0;
	MoveL Offs(p0,356.1,219.55, 0), v100, z5, tool0;
	MoveL Offs(p0,357.8016,217.5552, 0), v100, z5, tool0;
	MoveL Offs(p0,359.5368,216.0236, 0), v100, z5, tool0;
	MoveL Offs(p0,361.2912,214.9744, 0), v100, z5, tool0;
	MoveL Offs(p0,363.05039999999997,214.42680000000001, 0), v100, z5, tool0;
	MoveL Offs(p0,364.8,214.4, 0), v100, z5, tool0;
	MoveL Offs(p0,367.4802,215.7122, 0), v100, z5, tool0;
	MoveL Offs(p0,368.1184,216.7264, 0), v100, z5, tool0;
	MoveL Offs(p0,368.675,218.175, 0), v100, z5, tool0;
	MoveL Offs(p0,369.1776,220.1456, 0), v100, z5, tool0;
	MoveL Offs(p0,369.6538,222.7258, 0), v100, z5, tool0;
	MoveL Offs(p0,370.1312000000001,226.00320000000002, 0), v100, z5, tool0;
	MoveL Offs(p0,370.63739999999996,230.06540000000004, 0), v100, z5, tool0;
	MoveL Offs(p0,371.2,235.0, 0), v100, z5, tool0;
	MoveL Offs(p0,371.5708000000001,238.30300000000003, 0), v100, z5, tool0;
	MoveL Offs(p0,371.9584000000001,241.57600000000008, 0), v100, z5, tool0;
	MoveL Offs(p0,372.3556,244.76499999999996, 0), v100, z5, tool0;
	MoveL Offs(p0,372.75520000000006,247.81600000000003, 0), v100, z5, tool0;
	MoveL Offs(p0,373.15,250.675, 0), v100, z5, tool0;
	MoveL Offs(p0,373.53279999999995,253.288, 0), v100, z5, tool0;
	MoveL Offs(p0,373.89639999999997,255.60100000000003, 0), v100, z5, tool0;
	MoveL Offs(p0,374.2336,257.56000000000006, 0), v100, z5, tool0;
	MoveL Offs(p0,374.53720000000004,259.111, 0), v100, z5, tool0;
	MoveL Offs(p0,374.8,260.2, 0), v100, z5, tool0;
	MoveL Offs(p0,376.2,265.4, 0), v100, z5, tool0;
	MoveL Offs(p0,388.8,261.2, 0), v100, z5, tool0;
	MoveL Offs(p0,401.6,257.2, 0), v100, z5, tool0;
	MoveL Offs(p0,397.8,250.0, 0), v100, z5, tool0;
	MoveL Offs(p0,395.3350000000001,244.31640000000002, 0), v100, z5, tool0;
	MoveL Offs(p0,393.3440000000001,237.7232, 0), v100, z5, tool0;
	MoveL Offs(p0,391.833,230.42679999999996, 0), v100, z5, tool0;
	MoveL Offs(p0,390.808,222.63360000000003, 0), v100, z5, tool0;
	MoveL Offs(p0,390.275,214.55, 0), v100, z5, tool0;
	MoveL Offs(p0,390.24,206.38240000000002, 0), v100, z5, tool0;
	MoveL Offs(p0,390.709,198.3372, 0), v100, z5, tool0;
	MoveL Offs(p0,391.688,190.6208, 0), v100, z5, tool0;
	MoveL Offs(p0,393.183,183.4396, 0), v100, z5, tool0;
	MoveL Offs(p0,395.2,177.0, 0), v100, z5, tool0;
	MoveL Offs(p0,396.02979999999997,174.6168, 0), v100, z5, tool0;
	MoveL Offs(p0,395.9616,174.2896, 0), v100, z5, tool0;
	MoveL Offs(p0,395.675,174.2, 0), v100, z5, tool0;
	MoveL Offs(p0,395.1424,174.35039999999998, 0), v100, z5, tool0;
	MoveL Offs(p0,394.3362,174.7432, 0), v100, z5, tool0;
	MoveL Offs(p0,391.79260000000005,176.2656, 0), v100, z5, tool0;
	MoveL Offs(p0,390.0,177.4, 0), v100, z5, tool0;
	MoveL Offs(p0,380.8652000000001,183.80480000000003, 0), v100, z5, tool0;
	MoveL Offs(p0,372.45760000000007,190.95840000000004, 0), v100, z5, tool0;
	MoveL Offs(p0,364.8324,198.7696, 0), v100, z5, tool0;
	MoveL Offs(p0,358.0448,207.14720000000005, 0), v100, z5, tool0;
	MoveL Offs(p0,352.15,216.0, 0), v100, z5, tool0;
	MoveL Offs(p0,347.20320000000004,225.23680000000004, 0), v100, z5, tool0;
	MoveL Offs(p0,343.2596,234.76640000000003, 0), v100, z5, tool0;
	MoveL Offs(p0,340.37440000000004,244.49760000000006, 0), v100, z5, tool0;
	MoveL Offs(p0,338.6028,254.33920000000003, 0), v100, z5, tool0;
	MoveL Offs(p0,338.0,264.2, 0), v100, z5, tool0;
	MoveL Offs(p0,338.09900000000005,269.1342000000001, 0), v100, z5, tool0;
	MoveL Offs(p0,338.38400000000007,273.6976000000001, 0), v100, z5, tool0;
	MoveL Offs(p0,338.837,277.8314, 0), v100, z5, tool0;
	MoveL Offs(p0,339.43999999999994,281.4768, 0), v100, z5, tool0;
	MoveL Offs(p0,340.175,284.575, 0), v100, z5, tool0;
	MoveL Offs(p0,341.024,287.0672, 0), v100, z5, tool0;
	MoveL Offs(p0,341.96899999999994,288.89459999999997, 0), v100, z5, tool0;
	MoveL Offs(p0,342.992,289.99840000000006, 0), v100, z5, tool0;
	MoveL Offs(p0,344.075,290.31980000000004, 0), v100, z5, tool0;
	MoveL Offs(p0,345.2,289.8, 0), v100, z5, tool0;
	MoveL Offs(p0,346.5356,287.09099999999995, 0), v100, z5, tool0;
	MoveL Offs(p0,346.78720000000004,285.544, 0), v100, z5, tool0;
	MoveL Offs(p0,346.95,283.625, 0), v100, z5, tool0;
	MoveL Offs(p0,347.0288,281.304, 0), v100, z5, tool0;
	MoveL Offs(p0,347.02840000000003,278.55100000000004, 0), v100, z5, tool0;
	MoveL Offs(p0,346.9536,275.33600000000007, 0), v100, z5, tool0;
	MoveL Offs(p0,346.80920000000003,271.629, 0), v100, z5, tool0;
	MoveL Offs(p0,346.6,267.4, 0), v100, z5, tool0;
	MoveL Offs(p0,346.6,267.4, 0), v100, z5, tool0;
	MoveJ Offs(p0,525.4,287.0, 10), v100, z1, tool0;
	MoveL Offs(p0,527.7946000000002,284.4100000000001, 0), v100, z5, tool0;
	MoveL Offs(p0,529.9168000000002,280.39200000000005, 0), v100, z5, tool0;
	MoveL Offs(p0,531.7342,275.17400000000004, 0), v100, z5, tool0;
	MoveL Offs(p0,533.2144000000001,268.98400000000004, 0), v100, z5, tool0;
	MoveL Offs(p0,534.325,262.05, 0), v100, z5, tool0;
	MoveL Offs(p0,535.0336,254.6, 0), v100, z5, tool0;
	MoveL Offs(p0,535.3077999999999,246.862, 0), v100, z5, tool0;
	MoveL Offs(p0,535.1152,239.06400000000002, 0), v100, z5, tool0;
	MoveL Offs(p0,534.4234,231.43400000000003, 0), v100, z5, tool0;
	MoveL Offs(p0,533.2,224.2, 0), v100, z5, tool0;
	MoveL Offs(p0,531.4230000000001,217.05280000000002, 0), v100, z5, tool0;
	MoveL Offs(p0,529.2080000000003,210.36640000000006, 0), v100, z5, tool0;
	MoveL Offs(p0,526.549,204.1336, 0), v100, z5, tool0;
	MoveL Offs(p0,523.44,198.3472, 0), v100, z5, tool0;
	MoveL Offs(p0,519.875,193.0, 0), v100, z5, tool0;
	MoveL Offs(p0,515.848,188.0848, 0), v100, z5, tool0;
	MoveL Offs(p0,511.35299999999995,183.5944, 0), v100, z5, tool0;
	MoveL Offs(p0,506.384,179.5216, 0), v100, z5, tool0;
	MoveL Offs(p0,500.93500000000006,175.85920000000002, 0), v100, z5, tool0;
	MoveL Offs(p0,495.0,172.6, 0), v100, z5, tool0;
	MoveL Offs(p0,491.25960000000003,170.8452, 0), v100, z5, tool0;
	MoveL Offs(p0,487.0608000000001,169.19360000000003, 0), v100, z5, tool0;
	MoveL Offs(p0,482.49719999999996,167.66439999999997, 0), v100, z5, tool0;
	MoveL Offs(p0,477.66240000000005,166.27680000000004, 0), v100, z5, tool0;
	MoveL Offs(p0,472.65,165.05, 0), v100, z5, tool0;
	MoveL Offs(p0,467.5536,164.00320000000002, 0), v100, z5, tool0;
	MoveL Offs(p0,462.4668,163.1556, 0), v100, z5, tool0;
	MoveL Offs(p0,457.4832,162.52640000000002, 0), v100, z5, tool0;
	MoveL Offs(p0,452.6964,162.1348, 0), v100, z5, tool0;
	MoveL Offs(p0,448.2,162.0, 0), v100, z5, tool0;
	MoveL Offs(p0,443.45340000000016,162.14960000000002, 0), v100, z5, tool0;
	MoveL Offs(p0,438.3312000000001,162.57280000000006, 0), v100, z5, tool0;
	MoveL Offs(p0,433.0098,163.2312, 0), v100, z5, tool0;
	MoveL Offs(p0,427.6656,164.0864, 0), v100, z5, tool0;
	MoveL Offs(p0,422.475,165.1, 0), v100, z5, tool0;
	MoveL Offs(p0,417.61439999999993,166.2336, 0), v100, z5, tool0;
	MoveL Offs(p0,413.2602,167.4488, 0), v100, z5, tool0;
	MoveL Offs(p0,409.5888,168.7072, 0), v100, z5, tool0;
	MoveL Offs(p0,406.77660000000003,169.9704, 0), v100, z5, tool0;
	MoveL Offs(p0,405.0,171.2, 0), v100, z5, tool0;
	MoveL Offs(p0,402.5208,174.7896, 0), v100, z5, tool0;
	MoveL Offs(p0,400.3824000000001,179.94880000000006, 0), v100, z5, tool0;
	MoveL Offs(p0,398.6136,186.36319999999998, 0), v100, z5, tool0;
	MoveL Offs(p0,397.2432,193.71840000000003, 0), v100, z5, tool0;
	MoveL Offs(p0,396.3,201.7, 0), v100, z5, tool0;
	MoveL Offs(p0,395.81280000000004,209.99360000000001, 0), v100, z5, tool0;
	MoveL Offs(p0,395.8104,218.2848, 0), v100, z5, tool0;
	MoveL Offs(p0,396.32160000000005,226.25920000000002, 0), v100, z5, tool0;
	MoveL Offs(p0,397.37520000000006,233.6024, 0), v100, z5, tool0;
	MoveL Offs(p0,399.0,240.0, 0), v100, z5, tool0;
	MoveL Offs(p0,400.36480000000006,243.91840000000002, 0), v100, z5, tool0;
	MoveL Offs(p0,401.68640000000016,247.08320000000003, 0), v100, z5, tool0;
	MoveL Offs(p0,403.12559999999996,249.5688, 0), v100, z5, tool0;
	MoveL Offs(p0,404.8432000000001,251.4496, 0), v100, z5, tool0;
	MoveL Offs(p0,407.0,252.8, 0), v100, z5, tool0;
	MoveL Offs(p0,409.7568,253.6944, 0), v100, z5, tool0;
	MoveL Offs(p0,413.27439999999996,254.2072, 0), v100, z5, tool0;
	MoveL Offs(p0,417.71360000000004,254.4128, 0), v100, z5, tool0;
	MoveL Offs(p0,423.23519999999996,254.38559999999998, 0), v100, z5, tool0;
	MoveL Offs(p0,430.0,254.2, 0), v100, z5, tool0;
	MoveL Offs(p0,433.67300000000006,254.1694, 0), v100, z5, tool0;
	MoveL Offs(p0,437.44800000000015,254.19520000000006, 0), v100, z5, tool0;
	MoveL Offs(p0,441.259,254.2738, 0), v100, z5, tool0;
	MoveL Offs(p0,445.0400000000001,254.40160000000006, 0), v100, z5, tool0;
	MoveL Offs(p0,448.725,254.575, 0), v100, z5, tool0;
	MoveL Offs(p0,452.24799999999993,254.79039999999995, 0), v100, z5, tool0;
	MoveL Offs(p0,455.543,255.0442, 0), v100, z5, tool0;
	MoveL Offs(p0,458.54400000000004,255.33280000000005, 0), v100, z5, tool0;
	MoveL Offs(p0,461.18500000000006,255.65259999999998, 0), v100, z5, tool0;
	MoveL Offs(p0,463.4,256.0, 0), v100, z5, tool0;
	MoveL Offs(p0,468.57600000000014,257.2442, 0), v100, z5, tool0;
	MoveL Offs(p0,473.7520000000001,258.8016000000001, 0), v100, z5, tool0;
	MoveL Offs(p0,478.88,260.64939999999996, 0), v100, z5, tool0;
	MoveL Offs(p0,483.9120000000001,262.76480000000004, 0), v100, z5, tool0;
	MoveL Offs(p0,488.8,265.125, 0), v100, z5, tool0;
	MoveL Offs(p0,493.4959999999999,267.7072, 0), v100, z5, tool0;
	MoveL Offs(p0,497.95199999999994,270.4886, 0), v100, z5, tool0;
	MoveL Offs(p0,502.12000000000006,273.4464, 0), v100, z5, tool0;
	MoveL Offs(p0,505.95200000000006,276.5578, 0), v100, z5, tool0;
	MoveL Offs(p0,509.4,279.8, 0), v100, z5, tool0;
	MoveL Offs(p0,512.4416000000001,282.8944000000001, 0), v100, z5, tool0;
	MoveL Offs(p0,513.8693999999999,284.3036, 0), v100, z5, tool0;
	MoveL Offs(p0,515.2048000000001,285.59520000000003, 0), v100, z5, tool0;
	MoveL Offs(p0,516.425,286.75, 0), v100, z5, tool0;
	MoveL Offs(p0,517.5072,287.74879999999996, 0), v100, z5, tool0;
	MoveL Offs(p0,518.4286,288.57239999999996, 0), v100, z5, tool0;
	MoveL Offs(p0,519.1664000000001,289.2016, 0), v100, z5, tool0;
	MoveL Offs(p0,519.6978,289.6172, 0), v100, z5, tool0;
	MoveL Offs(p0,520.0,289.8, 0), v100, z5, tool0;
	MoveL Offs(p0,522.025,289.075, 0), v100, z5, tool0;
	MoveL Offs(p0,522.6351999999999,288.7344, 0), v100, z5, tool0;
	MoveL Offs(p0,523.2886,288.3482, 0), v100, z5, tool0;
	MoveL Offs(p0,523.9744000000001,287.9248, 0), v100, z5, tool0;
	MoveL Offs(p0,524.6818000000001,287.47260000000006, 0), v100, z5, tool0;
	MoveL Offs(p0,525.4,287.0, 0), v100, z5, tool0;
	MoveL Offs(p0,525.4,287.0, 0), v100, z5, tool0;
	MoveJ Offs(p0,370.6,255.4, 10), v100, z1, tool0;
	MoveL Offs(p0,370.187,253.2544000000001, 0), v100, z5, tool0;
	MoveL Offs(p0,369.7920000000001,250.93120000000008, 0), v100, z5, tool0;
	MoveL Offs(p0,369.421,248.4808, 0), v100, z5, tool0;
	MoveL Offs(p0,369.08000000000004,245.9536, 0), v100, z5, tool0;
	MoveL Offs(p0,368.775,243.4, 0), v100, z5, tool0;
	MoveL Offs(p0,368.51200000000006,240.87040000000002, 0), v100, z5, tool0;
	MoveL Offs(p0,368.29699999999997,238.4152, 0), v100, z5, tool0;
	MoveL Offs(p0,368.1360000000001,236.0848, 0), v100, z5, tool0;
	MoveL Offs(p0,368.035,233.92960000000002, 0), v100, z5, tool0;
	MoveL Offs(p0,368.0,232.0, 0), v100, z5, tool0;
	MoveL Offs(p0,367.93820000000005,228.16800000000003, 0), v100, z5, tool0;
	MoveL Offs(p0,367.7456000000001,224.93600000000006, 0), v100, z5, tool0;
	MoveL Offs(p0,367.4114,222.28000000000003, 0), v100, z5, tool0;
	MoveL Offs(p0,366.92480000000006,220.17600000000002, 0), v100, z5, tool0;
	MoveL Offs(p0,366.275,218.6, 0), v100, z5, tool0;
	MoveL Offs(p0,365.4512,217.52800000000002, 0), v100, z5, tool0;
	MoveL Offs(p0,364.44259999999997,216.936, 0), v100, z5, tool0;
	MoveL Offs(p0,363.2384,216.8, 0), v100, z5, tool0;
	MoveL Offs(p0,361.8278,217.096, 0), v100, z5, tool0;
	MoveL Offs(p0,360.2,217.8, 0), v100, z5, tool0;
	MoveL Offs(p0,357.809,220.05640000000002, 0), v100, z5, tool0;
	MoveL Offs(p0,355.59200000000016,223.97120000000004, 0), v100, z5, tool0;
	MoveL Offs(p0,353.60299999999995,229.2228, 0), v100, z5, tool0;
	MoveL Offs(p0,351.896,235.48960000000002, 0), v100, z5, tool0;
	MoveL Offs(p0,350.525,242.45, 0), v100, z5, tool0;
	MoveL Offs(p0,349.544,249.7824, 0), v100, z5, tool0;
	MoveL Offs(p0,349.00699999999995,257.1652, 0), v100, z5, tool0;
	MoveL Offs(p0,348.968,264.2768, 0), v100, z5, tool0;
	MoveL Offs(p0,349.481,270.79560000000004, 0), v100, z5, tool0;
	MoveL Offs(p0,350.6,276.4, 0), v100, z5, tool0;
	MoveL Offs(p0,352.0,282.0, 0), v100, z5, tool0;
	MoveL Offs(p0,362.6,275.0, 0), v100, z5, tool0;
	MoveL Offs(p0,373.4,267.8, 0), v100, z5, tool0;
	MoveL Offs(p0,370.6,255.4, 0), v100, z5, tool0;
	MoveL Offs(p0,370.6,255.4, 0), v100, z5, tool0;
	MoveJ Offs(p0,92.6,259.4, 10), v100, z1, tool0;
	MoveL Offs(p0,95.19700000000002,257.82340000000005, 0), v100, z5, tool0;
	MoveL Offs(p0,97.24800000000003,256.48320000000007, 0), v100, z5, tool0;
	MoveL Offs(p0,98.78299999999999,255.24380000000002, 0), v100, z5, tool0;
	MoveL Offs(p0,99.83200000000001,253.96960000000004, 0), v100, z5, tool0;
	MoveL Offs(p0,100.425,252.525, 0), v100, z5, tool0;
	MoveL Offs(p0,100.592,250.7744, 0), v100, z5, tool0;
	MoveL Offs(p0,100.36299999999999,248.5822, 0), v100, z5, tool0;
	MoveL Offs(p0,99.768,245.81280000000007, 0), v100, z5, tool0;
	MoveL Offs(p0,98.83700000000002,242.3306, 0), v100, z5, tool0;
	MoveL Offs(p0,97.6,238.0, 0), v100, z5, tool0;
	MoveL Offs(p0,96.35760000000002,233.65720000000005, 0), v100, z5, tool0;
	MoveL Offs(p0,95.22080000000003,230.04160000000007, 0), v100, z5, tool0;
	MoveL Offs(p0,94.1152,227.05239999999995, 0), v100, z5, tool0;
	MoveL Offs(p0,92.96640000000001,224.5888, 0), v100, z5, tool0;
	MoveL Offs(p0,91.7,222.55, 0), v100, z5, tool0;
	MoveL Offs(p0,90.24159999999999,220.8352, 0), v100, z5, tool0;
	MoveL Offs(p0,88.5168,219.34359999999998, 0), v100, z5, tool0;
	MoveL Offs(p0,86.4512,217.9744, 0), v100, z5, tool0;
	MoveL Offs(p0,83.97040000000001,216.6268, 0), v100, z5, tool0;
	MoveL Offs(p0,81.0,215.2, 0), v100, z5, tool0;
	MoveL Offs(p0,77.11840000000004,213.27200000000008, 0), v100, z5, tool0;
	MoveL Offs(p0,75.02759999999999,212.077, 0), v100, z5, tool0;
	MoveL Offs(p0,72.89120000000001,210.76800000000003, 0), v100, z5, tool0;
	MoveL Offs(p0,70.75,209.375, 0), v100, z5, tool0;
	MoveL Offs(p0,68.64479999999999,207.92800000000003, 0), v100, z5, tool0;
	MoveL Offs(p0,66.6164,206.45700000000002, 0), v100, z5, tool0;
	MoveL Offs(p0,64.7056,204.99200000000002, 0), v100, z5, tool0;
	MoveL Offs(p0,62.9532,203.56300000000002, 0), v100, z5, tool0;
	MoveL Offs(p0,61.4,202.2, 0), v100, z5, tool0;
	MoveL Offs(p0,52.4,193.8, 0), v100, z5, tool0;
	MoveL Offs(p0,47.2,202.8, 0), v100, z5, tool0;
	MoveL Offs(p0,44.782000000000004,206.8442, 0), v100, z5, tool0;
	MoveL Offs(p0,42.448000000000015,210.45760000000004, 0), v100, z5, tool0;
	MoveL Offs(p0,40.19799999999999,213.64139999999998, 0), v100, z5, tool0;
	MoveL Offs(p0,38.032,216.39680000000004, 0), v100, z5, tool0;
	MoveL Offs(p0,35.95,218.725, 0), v100, z5, tool0;
	MoveL Offs(p0,33.952,220.6272, 0), v100, z5, tool0;
	MoveL Offs(p0,32.038,222.10460000000003, 0), v100, z5, tool0;
	MoveL Offs(p0,30.208000000000006,223.15840000000003, 0), v100, z5, tool0;
	MoveL Offs(p0,28.462,223.7898, 0), v100, z5, tool0;
	MoveL Offs(p0,26.8,224.0, 0), v100, z5, tool0;
	MoveL Offs(p0,24.611200000000004,223.84640000000007, 0), v100, z5, tool0;
	MoveL Offs(p0,23.822799999999997,223.58959999999996, 0), v100, z5, tool0;
	MoveL Offs(p0,23.209600000000002,223.1552, 0), v100, z5, tool0;
	MoveL Offs(p0,22.75,222.5, 0), v100, z5, tool0;
	MoveL Offs(p0,22.4224,221.5808, 0), v100, z5, tool0;
	MoveL Offs(p0,22.2052,220.3544, 0), v100, z5, tool0;
	MoveL Offs(p0,22.076800000000002,218.77759999999998, 0), v100, z5, tool0;
	MoveL Offs(p0,22.0156,216.80720000000002, 0), v100, z5, tool0;
	MoveL Offs(p0,22.0,214.4, 0), v100, z5, tool0;
	MoveL Offs(p0,22.136600000000005,210.6368, 0), v100, z5, tool0;
	MoveL Offs(p0,22.540800000000008,206.68640000000005, 0), v100, z5, tool0;
	MoveL Offs(p0,23.204199999999997,202.5776, 0), v100, z5, tool0;
	MoveL Offs(p0,24.1184,198.33920000000003, 0), v100, z5, tool0;
	MoveL Offs(p0,25.275,194.0, 0), v100, z5, tool0;
	MoveL Offs(p0,26.6656,189.5888, 0), v100, z5, tool0;
	MoveL Offs(p0,28.281799999999997,185.13439999999997, 0), v100, z5, tool0;
	MoveL Offs(p0,30.115200000000005,180.6656, 0), v100, z5, tool0;
	MoveL Offs(p0,32.1574,176.21120000000002, 0), v100, z5, tool0;
	MoveL Offs(p0,34.4,171.8, 0), v100, z5, tool0;
	MoveL Offs(p0,36.20800000000001,168.00480000000005, 0), v100, z5, tool0;
	MoveL Offs(p0,37.010000000000005,166.1012, 0), v100, z5, tool0;
	MoveL Offs(p0,37.728,164.2384, 0), v100, z5, tool0;
	MoveL Offs(p0,38.35,162.45, 0), v100, z5, tool0;
	MoveL Offs(p0,38.864,160.7696, 0), v100, z5, tool0;
	MoveL Offs(p0,39.257999999999996,159.2308, 0), v100, z5, tool0;
	MoveL Offs(p0,39.52,157.8672, 0), v100, z5, tool0;
	MoveL Offs(p0,39.638,156.7124, 0), v100, z5, tool0;
	MoveL Offs(p0,39.6,155.8, 0), v100, z5, tool0;
	MoveL Offs(p0,38.8818,153.4078, 0), v100, z5, tool0;
	MoveL Offs(p0,38.48960000000001,153.2816, 0), v100, z5, tool0;
	MoveL Offs(p0,37.975,153.525, 0), v100, z5, tool0;
	MoveL Offs(p0,37.3104,154.1584, 0), v100, z5, tool0;
	MoveL Offs(p0,36.468199999999996,155.2022, 0), v100, z5, tool0;
	MoveL Offs(p0,35.4208,156.67680000000001, 0), v100, z5, tool0;
	MoveL Offs(p0,34.1406,158.6026, 0), v100, z5, tool0;
	MoveL Offs(p0,32.6,161.0, 0), v100, z5, tool0;
	MoveL Offs(p0,30.304400000000005,164.82800000000003, 0), v100, z5, tool0;
	MoveL Offs(p0,28.107200000000006,168.84800000000004, 0), v100, z5, tool0;
	MoveL Offs(p0,26.0228,173.024, 0), v100, z5, tool0;
	MoveL Offs(p0,24.065600000000003,177.32000000000002, 0), v100, z5, tool0;
	MoveL Offs(p0,22.25,181.7, 0), v100, z5, tool0;
	MoveL Offs(p0,20.590399999999995,186.12800000000001, 0), v100, z5, tool0;
	MoveL Offs(p0,19.1012,190.568, 0), v100, z5, tool0;
	MoveL Offs(p0,17.7968,194.984, 0), v100, z5, tool0;
	MoveL Offs(p0,16.6916,199.34, 0), v100, z5, tool0;
	MoveL Offs(p0,15.8,203.6, 0), v100, z5, tool0;
	MoveL Offs(p0,14.9364,210.519, 0), v100, z5, tool0;
	MoveL Offs(p0,14.963200000000004,217.31200000000004, 0), v100, z5, tool0;
	MoveL Offs(p0,15.846800000000002,223.91299999999995, 0), v100, z5, tool0;
	MoveL Offs(p0,17.5536,230.25600000000003, 0), v100, z5, tool0;
	MoveL Offs(p0,20.05,236.275, 0), v100, z5, tool0;
	MoveL Offs(p0,23.302400000000002,241.904, 0), v100, z5, tool0;
	MoveL Offs(p0,27.277200000000004,247.077, 0), v100, z5, tool0;
	MoveL Offs(p0,31.940800000000007,251.728, 0), v100, z5, tool0;
	MoveL Offs(p0,37.259600000000006,255.791, 0), v100, z5, tool0;
	MoveL Offs(p0,43.2,259.2, 0), v100, z5, tool0;
	MoveL Offs(p0,48.951800000000006,261.79760000000005, 0), v100, z5, tool0;
	MoveL Offs(p0,54.36640000000002,263.82880000000006, 0), v100, z5, tool0;
	MoveL Offs(p0,59.50260000000001,265.2912, 0), v100, z5, tool0;
	MoveL Offs(p0,64.4192,266.18240000000003, 0), v100, z5, tool0;
	MoveL Offs(p0,69.175,266.5, 0), v100, z5, tool0;
	MoveL Offs(p0,73.8288,266.2416, 0), v100, z5, tool0;
	MoveL Offs(p0,78.4394,265.40479999999997, 0), v100, z5, tool0;
	MoveL Offs(p0,83.06560000000002,263.98720000000003, 0), v100, z5, tool0;
	MoveL Offs(p0,87.7662,261.98640000000006, 0), v100, z5, tool0;
	MoveL Offs(p0,92.6,259.4, 0), v100, z5, tool0;
	MoveL Offs(p0,92.6,259.4, 0), v100, z5, tool0;
	MoveJ Offs(p0,341.4,221.4, 10), v100, z1, tool0;
	MoveL Offs(p0,342.1504000000001,219.30560000000006, 0), v100, z5, tool0;
	MoveL Offs(p0,342.2586,218.3364, 0), v100, z5, tool0;
	MoveL Offs(p0,342.17120000000006,217.3648, 0), v100, z5, tool0;
	MoveL Offs(p0,341.875,216.35, 0), v100, z5, tool0;
	MoveL Offs(p0,341.35679999999996,215.2512, 0), v100, z5, tool0;
	MoveL Offs(p0,340.60339999999997,214.02759999999998, 0), v100, z5, tool0;
	MoveL Offs(p0,339.6016000000001,212.6384, 0), v100, z5, tool0;
	MoveL Offs(p0,338.33820000000003,211.0428, 0), v100, z5, tool0;
	MoveL Offs(p0,336.8,209.2, 0), v100, z5, tool0;
	MoveL Offs(p0,332.01660000000004,202.57780000000002, 0), v100, z5, tool0;
	MoveL Offs(p0,328.1248000000001,195.07840000000004, 0), v100, z5, tool0;
	MoveL Offs(p0,325.1522,187.0726, 0), v100, z5, tool0;
	MoveL Offs(p0,323.1264,178.93120000000002, 0), v100, z5, tool0;
	MoveL Offs(p0,322.075,171.025, 0), v100, z5, tool0;
	MoveL Offs(p0,322.0256,163.72480000000002, 0), v100, z5, tool0;
	MoveL Offs(p0,323.0058,157.4014, 0), v100, z5, tool0;
	MoveL Offs(p0,325.0432,152.42560000000003, 0), v100, z5, tool0;
	MoveL Offs(p0,328.16540000000003,149.1682, 0), v100, z5, tool0;
	MoveL Offs(p0,332.4,148.0, 0), v100, z5, tool0;
	MoveL Offs(p0,334.40960000000007,148.67360000000005, 0), v100, z5, tool0;
	MoveL Offs(p0,335.80740000000003,149.49039999999997, 0), v100, z5, tool0;
	MoveL Offs(p0,337.43680000000006,150.6048, 0), v100, z5, tool0;
	MoveL Offs(p0,339.275,152.0, 0), v100, z5, tool0;
	MoveL Offs(p0,341.29920000000004,153.6592, 0), v100, z5, tool0;
	MoveL Offs(p0,343.4866,155.5656, 0), v100, z5, tool0;
	MoveL Offs(p0,345.81440000000003,157.7024, 0), v100, z5, tool0;
	MoveL Offs(p0,348.2598,160.0528, 0), v100, z5, tool0;
	MoveL Offs(p0,350.8,162.6, 0), v100, z5, tool0;
	MoveL Offs(p0,356.44480000000004,168.47600000000003, 0), v100, z5, tool0;
	MoveL Offs(p0,360.94240000000013,173.08000000000004, 0), v100, z5, tool0;
	MoveL Offs(p0,364.53759999999994,176.496, 0), v100, z5, tool0;
	MoveL Offs(p0,367.4752,178.80800000000002, 0), v100, z5, tool0;
	MoveL Offs(p0,370.0,180.1, 0), v100, z5, tool0;
	MoveL Offs(p0,372.3568,180.45600000000002, 0), v100, z5, tool0;
	MoveL Offs(p0,374.7904,179.95999999999998, 0), v100, z5, tool0;
	MoveL Offs(p0,377.54560000000004,178.696, 0), v100, z5, tool0;
	MoveL Offs(p0,380.8672,176.748, 0), v100, z5, tool0;
	MoveL Offs(p0,385.0,174.2, 0), v100, z5, tool0;
	MoveL Offs(p0,398.4,166.2, 0), v100, z5, tool0;
	MoveL Offs(p0,391.0,163.2, 0), v100, z5, tool0;
	MoveL Offs(p0,388.52800000000013,162.17600000000004, 0), v100, z5, tool0;
	MoveL Offs(p0,387.35499999999996,161.71499999999997, 0), v100, z5, tool0;
	MoveL Offs(p0,386.248,161.296, 0), v100, z5, tool0;
	MoveL Offs(p0,385.225,160.925, 0), v100, z5, tool0;
	MoveL Offs(p0,384.304,160.608, 0), v100, z5, tool0;
	MoveL Offs(p0,383.503,160.351, 0), v100, z5, tool0;
	MoveL Offs(p0,382.84000000000003,160.16, 0), v100, z5, tool0;
	MoveL Offs(p0,382.33299999999997,160.041, 0), v100, z5, tool0;
	MoveL Offs(p0,382.0,160.0, 0), v100, z5, tool0;
	MoveL Offs(p0,379.20640000000003,157.952, 0), v100, z5, tool0;
	MoveL Offs(p0,378.1,156.9, 0), v100, z5, tool0;
	MoveL Offs(p0,376.8736,155.68, 0), v100, z5, tool0;
	MoveL Offs(p0,375.54879999999997,154.316, 0), v100, z5, tool0;
	MoveL Offs(p0,374.14720000000005,152.83200000000002, 0), v100, z5, tool0;
	MoveL Offs(p0,372.6904,151.252, 0), v100, z5, tool0;
	MoveL Offs(p0,371.2,149.6, 0), v100, z5, tool0;
	MoveL Offs(p0,367.9216,145.5474, 0), v100, z5, tool0;
	MoveL Offs(p0,364.94080000000014,141.22720000000007, 0), v100, z5, tool0;
	MoveL Offs(p0,362.2792,136.6958, 0), v100, z5, tool0;
	MoveL Offs(p0,359.95840000000004,132.00960000000003, 0), v100, z5, tool0;
	MoveL Offs(p0,358.0,127.225, 0), v100, z5, tool0;
	MoveL Offs(p0,356.4256,122.3984, 0), v100, z5, tool0;
	MoveL Offs(p0,355.2568,117.5862, 0), v100, z5, tool0;
	MoveL Offs(p0,354.5152,112.8448, 0), v100, z5, tool0;
	MoveL Offs(p0,354.2224,108.23060000000001, 0), v100, z5, tool0;
	MoveL Offs(p0,354.4,103.8, 0), v100, z5, tool0;
	MoveL Offs(p0,354.6432000000001,100.70720000000003, 0), v100, z5, tool0;
	MoveL Offs(p0,354.6808,99.30179999999999, 0), v100, z5, tool0;
	MoveL Offs(p0,354.66560000000004,98.0176, 0), v100, z5, tool0;
	MoveL Offs(p0,354.6,96.875, 0), v100, z5, tool0;
	MoveL Offs(p0,354.4864,95.89439999999999, 0), v100, z5, tool0;
	MoveL Offs(p0,354.3272,95.0962, 0), v100, z5, tool0;
	MoveL Offs(p0,354.12480000000005,94.5008, 0), v100, z5, tool0;
	MoveL Offs(p0,353.8816,94.1286, 0), v100, z5, tool0;
	MoveL Offs(p0,353.6,94.0, 0), v100, z5, tool0;
	MoveL Offs(p0,349.98720000000014,95.89920000000004, 0), v100, z5, tool0;
	MoveL Offs(p0,347.3828,98.0608, 0), v100, z5, tool0;
	MoveL Offs(p0,344.42560000000003,100.8416, 0), v100, z5, tool0;
	MoveL Offs(p0,341.25,104.1, 0), v100, z5, tool0;
	MoveL Offs(p0,337.9904,107.6944, 0), v100, z5, tool0;
	MoveL Offs(p0,334.7812,111.48319999999998, 0), v100, z5, tool0;
	MoveL Offs(p0,331.7568,115.32480000000001, 0), v100, z5, tool0;
	MoveL Offs(p0,329.0516,119.0776, 0), v100, z5, tool0;
	MoveL Offs(p0,326.8,122.6, 0), v100, z5, tool0;
	MoveL Offs(p0,324.206,127.263, 0), v100, z5, tool0;
	MoveL Offs(p0,321.93600000000004,131.92000000000004, 0), v100, z5, tool0;
	MoveL Offs(p0,319.978,136.613, 0), v100, z5, tool0;
	MoveL Offs(p0,318.32000000000005,141.38400000000004, 0), v100, z5, tool0;
	MoveL Offs(p0,316.95,146.275, 0), v100, z5, tool0;
	MoveL Offs(p0,315.856,151.328, 0), v100, z5, tool0;
	MoveL Offs(p0,315.026,156.58499999999998, 0), v100, z5, tool0;
	MoveL Offs(p0,314.44800000000004,162.08800000000002, 0), v100, z5, tool0;
	MoveL Offs(p0,314.11,167.87900000000002, 0), v100, z5, tool0;
	MoveL Offs(p0,314.0,174.0, 0), v100, z5, tool0;
	MoveL Offs(p0,314.13480000000004,179.55800000000005, 0), v100, z5, tool0;
	MoveL Offs(p0,314.5504000000001,184.74400000000006, 0), v100, z5, tool0;
	MoveL Offs(p0,315.2636,189.606, 0), v100, z5, tool0;
	MoveL Offs(p0,316.2912,194.192, 0), v100, z5, tool0;
	MoveL Offs(p0,317.65,198.55, 0), v100, z5, tool0;
	MoveL Offs(p0,319.3568,202.728, 0), v100, z5, tool0;
	MoveL Offs(p0,321.42839999999995,206.77399999999997, 0), v100, z5, tool0;
	MoveL Offs(p0,323.88160000000005,210.73600000000002, 0), v100, z5, tool0;
	MoveL Offs(p0,326.7332,214.66200000000003, 0), v100, z5, tool0;
	MoveL Offs(p0,330.0,218.6, 0), v100, z5, tool0;
	MoveL Offs(p0,332.09040000000005,220.93560000000008, 0), v100, z5, tool0;
	MoveL Offs(p0,333.8352000000001,222.78880000000004, 0), v100, z5, tool0;
	MoveL Offs(p0,335.28479999999996,224.1692, 0), v100, z5, tool0;
	MoveL Offs(p0,336.4896,225.0864, 0), v100, z5, tool0;
	MoveL Offs(p0,337.5,225.55, 0), v100, z5, tool0;
	MoveL Offs(p0,338.3664,225.56959999999998, 0), v100, z5, tool0;
	MoveL Offs(p0,339.13919999999996,225.15479999999997, 0), v100, z5, tool0;
	MoveL Offs(p0,339.8688,224.3152, 0), v100, z5, tool0;
	MoveL Offs(p0,340.60560000000004,223.06040000000002, 0), v100, z5, tool0;
	MoveL Offs(p0,341.4,221.4, 0), v100, z5, tool0;
	MoveL Offs(p0,341.4,221.4, 0), v100, z5, tool0;
	MoveJ Offs(p0,36.0,214.8, 10), v100, z1, tool0;
	MoveL Offs(p0,38.17600000000001,212.06240000000008, 0), v100, z5, tool0;
	MoveL Offs(p0,39.33,210.49259999999998, 0), v100, z5, tool0;
	MoveL Offs(p0,40.496,208.83520000000004, 0), v100, z5, tool0;
	MoveL Offs(p0,41.65,207.125, 0), v100, z5, tool0;
	MoveL Offs(p0,42.767999999999994,205.39679999999998, 0), v100, z5, tool0;
	MoveL Offs(p0,43.826,203.6854, 0), v100, z5, tool0;
	MoveL Offs(p0,44.800000000000004,202.02560000000003, 0), v100, z5, tool0;
	MoveL Offs(p0,45.666000000000004,200.4522, 0), v100, z5, tool0;
	MoveL Offs(p0,46.4,199.0, 0), v100, z5, tool0;
	MoveL Offs(p0,50.6,190.4, 0), v100, z5, tool0;
	MoveL Offs(p0,46.0,178.2, 0), v100, z5, tool0;
	MoveL Offs(p0,44.576000000000015,174.32000000000005, 0), v100, z5, tool0;
	MoveL Offs(p0,43.894,172.56599999999997, 0), v100, z5, tool0;
	MoveL Offs(p0,43.248000000000005,170.96800000000002, 0), v100, z5, tool0;
	MoveL Offs(p0,42.65,169.55, 0), v100, z5, tool0;
	MoveL Offs(p0,42.112,168.33599999999998, 0), v100, z5, tool0;
	MoveL Offs(p0,41.646,167.35, 0), v100, z5, tool0;
	MoveL Offs(p0,41.263999999999996,166.61600000000004, 0), v100, z5, tool0;
	MoveL Offs(p0,40.977999999999994,166.158, 0), v100, z5, tool0;
	MoveL Offs(p0,40.8,166.0, 0), v100, z5, tool0;
	MoveL Offs(p0,38.055,169.92580000000004, 0), v100, z5, tool0;
	MoveL Offs(p0,36.656000000000006,172.6176, 0), v100, z5, tool0;
	MoveL Offs(p0,35.125,175.775, 0), v100, z5, tool0;
	MoveL Offs(p0,33.528,179.2624, 0), v100, z5, tool0;
	MoveL Offs(p0,31.931,182.9442, 0), v100, z5, tool0;
	MoveL Offs(p0,30.4,186.6848, 0), v100, z5, tool0;
	MoveL Offs(p0,29.000999999999998,190.3486, 0), v100, z5, tool0;
	MoveL Offs(p0,27.8,193.8, 0), v100, z5, tool0;
	MoveL Offs(p0,26.540799999999997,197.79720000000003, 0), v100, z5, tool0;
	MoveL Offs(p0,25.526400000000006,201.80160000000006, 0), v100, z5, tool0;
	MoveL Offs(p0,24.761599999999994,205.71239999999997, 0), v100, z5, tool0;
	MoveL Offs(p0,24.251200000000004,209.4288, 0), v100, z5, tool0;
	MoveL Offs(p0,24.0,212.85, 0), v100, z5, tool0;
	MoveL Offs(p0,24.012800000000002,215.8752, 0), v100, z5, tool0;
	MoveL Offs(p0,24.294400000000003,218.4036, 0), v100, z5, tool0;
	MoveL Offs(p0,24.849600000000002,220.33440000000002, 0), v100, z5, tool0;
	MoveL Offs(p0,25.6832,221.5668, 0), v100, z5, tool0;
	MoveL Offs(p0,26.8,222.0, 0), v100, z5, tool0;
	MoveL Offs(p0,28.812400000000004,221.2008, 0), v100, z5, tool0;
	MoveL Offs(p0,29.692800000000005,220.61760000000004, 0), v100, z5, tool0;
	MoveL Offs(p0,30.65,219.9, 0), v100, z5, tool0;
	MoveL Offs(p0,31.667199999999998,219.06239999999997, 0), v100, z5, tool0;
	MoveL Offs(p0,32.7276,218.1192, 0), v100, z5, tool0;
	MoveL Offs(p0,33.8144,217.0848, 0), v100, z5, tool0;
	MoveL Offs(p0,34.91080000000001,215.97360000000003, 0), v100, z5, tool0;
	MoveL Offs(p0,36.0,214.8, 0), v100, z5, tool0;
	MoveL Offs(p0,36.0,214.8, 0), v100, z5, tool0;
	MoveJ Offs(p0,103.4,201.0, 10), v100, z1, tool0;
	MoveL Offs(p0,106.018,197.83140000000003, 0), v100, z5, tool0;
	MoveL Offs(p0,108.76800000000003,194.29920000000004, 0), v100, z5, tool0;
	MoveL Offs(p0,111.554,190.54379999999998, 0), v100, z5, tool0;
	MoveL Offs(p0,114.28000000000002,186.7056, 0), v100, z5, tool0;
	MoveL Offs(p0,116.85,182.925, 0), v100, z5, tool0;
	MoveL Offs(p0,119.16799999999998,179.34240000000003, 0), v100, z5, tool0;
	MoveL Offs(p0,121.138,176.0982, 0), v100, z5, tool0;
	MoveL Offs(p0,122.66400000000002,173.33280000000002, 0), v100, z5, tool0;
	MoveL Offs(p0,123.65,171.1866, 0), v100, z5, tool0;
	MoveL Offs(p0,124.0,169.8, 0), v100, z5, tool0;
	MoveL Offs(p0,121.65,167.35, 0), v100, z5, tool0;
	MoveL Offs(p0,120.7168,166.56, 0), v100, z5, tool0;
	MoveL Offs(p0,119.66839999999999,165.698, 0), v100, z5, tool0;
	MoveL Offs(p0,118.5216,164.776, 0), v100, z5, tool0;
	MoveL Offs(p0,117.2932,163.80599999999998, 0), v100, z5, tool0;
	MoveL Offs(p0,116.0,162.8, 0), v100, z5, tool0;
	MoveL Offs(p0,113.43040000000005,160.78720000000004, 0), v100, z5, tool0;
	MoveL Offs(p0,112.22359999999999,159.74179999999998, 0), v100, z5, tool0;
	MoveL Offs(p0,111.0912,158.69760000000002, 0), v100, z5, tool0;
	MoveL Offs(p0,110.05,157.675, 0), v100, z5, tool0;
	MoveL Offs(p0,109.11679999999998,156.6944, 0), v100, z5, tool0;
	MoveL Offs(p0,108.3084,155.7762, 0), v100, z5, tool0;
	MoveL Offs(p0,107.64160000000001,154.94080000000002, 0), v100, z5, tool0;
	MoveL Offs(p0,107.13320000000002,154.2086, 0), v100, z5, tool0;
	MoveL Offs(p0,106.8,153.6, 0), v100, z5, tool0;
	MoveL Offs(p0,105.67200000000003,151.46560000000005, 0), v100, z5, tool0;
	MoveL Offs(p0,104.91900000000001,150.77939999999998, 0), v100, z5, tool0;
	MoveL Offs(p0,104.06400000000001,150.3488, 0), v100, z5, tool0;
	MoveL Offs(p0,103.125,150.175, 0), v100, z5, tool0;
	MoveL Offs(p0,102.12,150.25920000000002, 0), v100, z5, tool0;
	MoveL Offs(p0,101.067,150.6026, 0), v100, z5, tool0;
	MoveL Offs(p0,99.98400000000001,151.2064, 0), v100, z5, tool0;
	MoveL Offs(p0,98.88900000000001,152.0718, 0), v100, z5, tool0;
	MoveL Offs(p0,97.8,153.2, 0), v100, z5, tool0;
	MoveL Offs(p0,95.81460000000001,155.23300000000003, 0), v100, z5, tool0;
	MoveL Offs(p0,93.10080000000002,157.53600000000006, 0), v100, z5, tool0;
	MoveL Offs(p0,89.8422,159.99499999999998, 0), v100, z5, tool0;
	MoveL Offs(p0,86.22240000000001,162.496, 0), v100, z5, tool0;
	MoveL Offs(p0,82.425,164.925, 0), v100, z5, tool0;
	MoveL Offs(p0,78.6336,167.168, 0), v100, z5, tool0;
	MoveL Offs(p0,75.0318,169.11100000000002, 0), v100, z5, tool0;
	MoveL Offs(p0,71.8032,170.64000000000001, 0), v100, z5, tool0;
	MoveL Offs(p0,69.1314,171.64100000000002, 0), v100, z5, tool0;
	MoveL Offs(p0,67.2,172.0, 0), v100, z5, tool0;
	MoveL Offs(p0,63.02759999999999,171.20480000000003, 0), v100, z5, tool0;
	MoveL Offs(p0,60.19680000000002,168.95040000000003, 0), v100, z5, tool0;
	MoveL Offs(p0,58.6572,165.43359999999998, 0), v100, z5, tool0;
	MoveL Offs(p0,58.358399999999996,160.8512, 0), v100, z5, tool0;
	MoveL Offs(p0,59.25,155.4, 0), v100, z5, tool0;
	MoveL Offs(p0,61.281600000000005,149.2768, 0), v100, z5, tool0;
	MoveL Offs(p0,64.4028,142.67839999999998, 0), v100, z5, tool0;
	MoveL Offs(p0,68.56320000000001,135.8016, 0), v100, z5, tool0;
	MoveL Offs(p0,73.7124,128.8432, 0), v100, z5, tool0;
	MoveL Offs(p0,79.8,122.0, 0), v100, z5, tool0;
	MoveL Offs(p0,82.2954,119.41060000000002, 0), v100, z5, tool0;
	MoveL Offs(p0,84.40320000000003,117.12480000000005, 0), v100, z5, tool0;
	MoveL Offs(p0,86.1558,115.08619999999999, 0), v100, z5, tool0;
	MoveL Offs(p0,87.58560000000001,113.2384, 0), v100, z5, tool0;
	MoveL Offs(p0,88.725,111.525, 0), v100, z5, tool0;
	MoveL Offs(p0,89.6064,109.8896, 0), v100, z5, tool0;
	MoveL Offs(p0,90.2622,108.27579999999998, 0), v100, z5, tool0;
	MoveL Offs(p0,90.7248,106.62720000000002, 0), v100, z5, tool0;
	MoveL Offs(p0,91.0266,104.8874, 0), v100, z5, tool0;
	MoveL Offs(p0,91.2,103.0, 0), v100, z5, tool0;
	MoveL Offs(p0,91.48320000000004,100.09120000000003, 0), v100, z5, tool0;
	MoveL Offs(p0,91.6518,98.4838, 0), v100, z5, tool0;
	MoveL Offs(p0,91.8336,96.8176, 0), v100, z5, tool0;
	MoveL Offs(p0,92.025,95.125, 0), v100, z5, tool0;
	MoveL Offs(p0,92.22240000000001,93.4384, 0), v100, z5, tool0;
	MoveL Offs(p0,92.4222,91.7902, 0), v100, z5, tool0;
	MoveL Offs(p0,92.6208,90.21280000000002, 0), v100, z5, tool0;
	MoveL Offs(p0,92.81460000000001,88.73859999999999, 0), v100, z5, tool0;
	MoveL Offs(p0,93.0,87.4, 0), v100, z5, tool0;
	MoveL Offs(p0,93.43680000000003,83.88160000000002, 0), v100, z5, tool0;
	MoveL Offs(p0,93.5112,82.68039999999999, 0), v100, z5, tool0;
	MoveL Offs(p0,93.47040000000001,81.81280000000001, 0), v100, z5, tool0;
	MoveL Offs(p0,93.3,81.25, 0), v100, z5, tool0;
	MoveL Offs(p0,92.9856,80.9632, 0), v100, z5, tool0;
	MoveL Offs(p0,92.5128,80.9236, 0), v100, z5, tool0;
	MoveL Offs(p0,91.8672,81.10240000000002, 0), v100, z5, tool0;
	MoveL Offs(p0,91.0344,81.47080000000001, 0), v100, z5, tool0;
	MoveL Offs(p0,90.0,82.0, 0), v100, z5, tool0;
	MoveL Offs(p0,86.72939999999998,84.30579999999999, 0), v100, z5, tool0;
	MoveL Offs(p0,85.1648,85.54560000000001, 0), v100, z5, tool0;
	MoveL Offs(p0,83.425,86.975, 0), v100, z5, tool0;
	MoveL Offs(p0,81.5472,88.5664, 0), v100, z5, tool0;
	MoveL Offs(p0,79.5686,90.29220000000001, 0), v100, z5, tool0;
	MoveL Offs(p0,77.52640000000001,92.12480000000001, 0), v100, z5, tool0;
	MoveL Offs(p0,75.45779999999999,94.0366, 0), v100, z5, tool0;
	MoveL Offs(p0,73.4,96.0, 0), v100, z5, tool0;
	MoveL Offs(p0,68.3356,101.02940000000002, 0), v100, z5, tool0;
	MoveL Offs(p0,63.820800000000006,106.16320000000003, 0), v100, z5, tool0;
	MoveL Offs(p0,59.8532,111.40979999999999, 0), v100, z5, tool0;
	MoveL Offs(p0,56.4304,116.7776, 0), v100, z5, tool0;
	MoveL Offs(p0,53.55,122.275, 0), v100, z5, tool0;
	MoveL Offs(p0,51.2096,127.91040000000001, 0), v100, z5, tool0;
	MoveL Offs(p0,49.4068,133.6922, 0), v100, z5, tool0;
	MoveL Offs(p0,48.1392,139.6288, 0), v100, z5, tool0;
	MoveL Offs(p0,47.404399999999995,145.7286, 0), v100, z5, tool0;
	MoveL Offs(p0,47.2,152.0, 0), v100, z5, tool0;
	MoveL Offs(p0,47.3284,156.99280000000005, 0), v100, z5, tool0;
	MoveL Offs(p0,47.723200000000006,161.67840000000004, 0), v100, z5, tool0;
	MoveL Offs(p0,48.3988,166.0976, 0), v100, z5, tool0;
	MoveL Offs(p0,49.369600000000005,170.29120000000003, 0), v100, z5, tool0;
	MoveL Offs(p0,50.65,174.3, 0), v100, z5, tool0;
	MoveL Offs(p0,52.2544,178.1648, 0), v100, z5, tool0;
	MoveL Offs(p0,54.197199999999995,181.9264, 0), v100, z5, tool0;
	MoveL Offs(p0,56.49280000000001,185.62560000000002, 0), v100, z5, tool0;
	MoveL Offs(p0,59.15560000000001,189.3032, 0), v100, z5, tool0;
	MoveL Offs(p0,62.2,193.0, 0), v100, z5, tool0;
	MoveL Offs(p0,64.69040000000001,195.67040000000003, 0), v100, z5, tool0;
	MoveL Offs(p0,67.53120000000001,198.35520000000005, 0), v100, z5, tool0;
	MoveL Offs(p0,70.61680000000001,200.9848, 0), v100, z5, tool0;
	MoveL Offs(p0,73.84160000000001,203.4896, 0), v100, z5, tool0;
	MoveL Offs(p0,77.1,205.8, 0), v100, z5, tool0;
	MoveL Offs(p0,80.2864,207.8464, 0), v100, z5, tool0;
	MoveL Offs(p0,83.2952,209.5592, 0), v100, z5, tool0;
	MoveL Offs(p0,86.02080000000001,210.86880000000002, 0), v100, z5, tool0;
	MoveL Offs(p0,88.3576,211.7056, 0), v100, z5, tool0;
	MoveL Offs(p0,90.2,212.0, 0), v100, z5, tool0;
	MoveL Offs(p0,92.91259999999998,210.75799999999998, 0), v100, z5, tool0;
	MoveL Offs(p0,94.15520000000001,209.85600000000005, 0), v100, z5, tool0;
	MoveL Offs(p0,95.525,208.75, 0), v100, z5, tool0;
	MoveL Offs(p0,96.99680000000001,207.464, 0), v100, z5, tool0;
	MoveL Offs(p0,98.5454,206.022, 0), v100, z5, tool0;
	MoveL Offs(p0,100.14560000000002,204.44800000000004, 0), v100, z5, tool0;
	MoveL Offs(p0,101.7722,202.76600000000002, 0), v100, z5, tool0;
	MoveL Offs(p0,103.4,201.0, 0), v100, z5, tool0;
	MoveL Offs(p0,103.4,201.0, 0), v100, z5, tool0;
	MoveJ Offs(p0,351.4,205.4, 10), v100, z1, tool0;
	MoveL Offs(p0,353.21760000000006,203.01120000000006, 0), v100, z5, tool0;
	MoveL Offs(p0,354.28540000000004,201.6848, 0), v100, z5, tool0;
	MoveL Offs(p0,355.4288,200.3056, 0), v100, z5, tool0;
	MoveL Offs(p0,356.625,198.9, 0), v100, z5, tool0;
	MoveL Offs(p0,357.85119999999995,197.49439999999998, 0), v100, z5, tool0;
	MoveL Offs(p0,359.0846,196.11520000000002, 0), v100, z5, tool0;
	MoveL Offs(p0,360.30240000000003,194.7888, 0), v100, z5, tool0;
	MoveL Offs(p0,361.4818,193.54160000000002, 0), v100, z5, tool0;
	MoveL Offs(p0,362.6,192.4, 0), v100, z5, tool0;
	MoveL Offs(p0,369.4,185.8, 0), v100, z5, tool0;
	MoveL Offs(p0,352.0,169.0, 0), v100, z5, tool0;
	MoveL Offs(p0,349.19320000000005,166.2398, 0), v100, z5, tool0;
	MoveL Offs(p0,346.44160000000005,163.62240000000003, 0), v100, z5, tool0;
	MoveL Offs(p0,343.7884,161.18259999999998, 0), v100, z5, tool0;
	MoveL Offs(p0,341.2768,158.95520000000002, 0), v100, z5, tool0;
	MoveL Offs(p0,338.95,156.975, 0), v100, z5, tool0;
	MoveL Offs(p0,336.85119999999995,155.2768, 0), v100, z5, tool0;
	MoveL Offs(p0,335.02360000000004,153.89540000000002, 0), v100, z5, tool0;
	MoveL Offs(p0,333.5104,152.86560000000003, 0), v100, z5, tool0;
	MoveL Offs(p0,332.3548,152.22220000000002, 0), v100, z5, tool0;
	MoveL Offs(p0,331.6,152.0, 0), v100, z5, tool0;
	MoveL Offs(p0,328.8376,153.0908, 0), v100, z5, tool0;
	MoveL Offs(p0,326.99680000000006,156.11840000000007, 0), v100, z5, tool0;
	MoveL Offs(p0,326.0272,160.7156, 0), v100, z5, tool0;
	MoveL Offs(p0,325.8784,166.5152, 0), v100, z5, tool0;
	MoveL Offs(p0,326.5,173.15, 0), v100, z5, tool0;
	MoveL Offs(p0,327.8416,180.2528, 0), v100, z5, tool0;
	MoveL Offs(p0,329.8528,187.4564, 0), v100, z5, tool0;
	MoveL Offs(p0,332.4832,194.39360000000002, 0), v100, z5, tool0;
	MoveL Offs(p0,335.68240000000003,200.6972, 0), v100, z5, tool0;
	MoveL Offs(p0,339.4,206.0, 0), v100, z5, tool0;
	MoveL Offs(p0,341.7724,208.79539999999997, 0), v100, z5, tool0;
	MoveL Offs(p0,342.53280000000007,209.5808, 0), v100, z5, tool0;
	MoveL Offs(p0,343.25,210.275, 0), v100, z5, tool0;
	MoveL Offs(p0,343.9072,210.8672, 0), v100, z5, tool0;
	MoveL Offs(p0,344.48760000000004,211.3466, 0), v100, z5, tool0;
	MoveL Offs(p0,344.97440000000006,211.70240000000004, 0), v100, z5, tool0;
	MoveL Offs(p0,345.35080000000005,211.92380000000003, 0), v100, z5, tool0;
	MoveL Offs(p0,345.6,212.0, 0), v100, z5, tool0;
	MoveL Offs(p0,347.9,210.05, 0), v100, z5, tool0;
	MoveL Offs(p0,348.552,209.2784, 0), v100, z5, tool0;
	MoveL Offs(p0,349.23999999999995,208.41320000000002, 0), v100, z5, tool0;
	MoveL Offs(p0,349.95200000000006,207.46880000000002, 0), v100, z5, tool0;
	MoveL Offs(p0,350.67600000000004,206.4596, 0), v100, z5, tool0;
	MoveL Offs(p0,351.4,205.4, 0), v100, z5, tool0;
	MoveL Offs(p0,351.4,205.4, 0), v100, z5, tool0;
	MoveJ Offs(p0,158.0,186.6, 10), v100, z1, tool0;
	MoveL Offs(p0,159.48960000000005,184.38720000000006, 0), v100, z5, tool0;
	MoveL Offs(p0,159.8234,183.4158, 0), v100, z5, tool0;
	MoveL Offs(p0,159.88479999999998,182.52960000000002, 0), v100, z5, tool0;
	MoveL Offs(p0,159.675,181.725, 0), v100, z5, tool0;
	MoveL Offs(p0,159.19519999999997,180.9984, 0), v100, z5, tool0;
